TYPE "UDT_Motion_Point_IAI"
VERSION : 0.1
// =================================================================================
// UDT_Recipe_Final.scl
// Version: Final
//
// Description:
// Final, definitive recipe structure based on deep code analysis.
// - Axis names and mapping are CORRECT.
// - Position names are simple and numeric (Position_01, Position_02, ...)
//   to provide a safe, 1-to-1 mapping with the axis driver's position array.
//   This structure can be used to build a descriptive HMI.
// =================================================================================
// =================================================================================
// BASE TYPES for Motion Points
// =================================================================================
   STRUCT
      Pos : Real;   //  Target Position (um/pulse)
      Vel : Int;   //  Target Velocity (mm/s or %)
   END_STRUCT;

END_TYPE

TYPE "UDT_Motion_Point_V90"
VERSION : 0.1
   STRUCT
      Pos : DInt;   //  Target Position (mm/deg)
      Vel : Int;   //  Target Velocity (mm/s or rpm)
   END_STRUCT;

END_TYPE

TYPE "UDT_Recipe_PressCurve"
VERSION : 0.1
// NOTE: UDT_Recipe_PressCurve and UDT_Recipe_ATEQ are assumed to exist from original project files.
// =================================================================================
// MAIN RECIPE UDT - FINAL VERSION
// =================================================================================
   STRUCT
      StartPos_UL : Real;
      StartPos_LL : Real;
      StartForce_UL : Real;
      StartForce_LL : Real;
      MiddlePos_UL : Real;
      MiddlePos_LL : Real;
      MiddleForce_UL : Real;
      MiddleForce_LL : Real;
      FinalPos_UL : Real;
      FinalPos_LL : Real;
      FinalForce_UL : Real;
      FinalForce_LL : Real;
      ProgramNum : Int;
   END_STRUCT;

END_TYPE

TYPE "UDT_Gripper_Fixture_Codes"
VERSION : 0.1
// =================================================================================
// OTHER UDTs (Grippers, Process, etc. - Unchanged from previous correct versions)
// =================================================================================
   STRUCT
      "JAW TOOLING LEFT" : String[128];
      "JAW TOOLING RIGHT" : String[128];
      "SHAFT CLAMPING LEFT" : String[128];
      "SHAFT CLAMPING RIGHT" : String[128];
   END_STRUCT;

END_TYPE

TYPE "UDT_IAI_Axis_Positions"
VERSION : 0.1
// =================================================================================
// POSITION SETS - Mirroring the Axis Driver's Position Array
// =================================================================================
   STRUCT
      Position : Array[1..20] of "UDT_Motion_Point_IAI";
   END_STRUCT;

END_TYPE

TYPE "UDT_V90_Axis_Positions"
VERSION : 0.1
   STRUCT
      Position : Array[1..20] of "UDT_Motion_Point_V90";
   END_STRUCT;

END_TYPE

TYPE "UDT_OP10_Recipe_type"
VERSION : 0.1
   STRUCT
      Header : Struct   // Information about recipe
         RecipeName : String[50];   // name of product
         RecipeID : USInt;   // number of product for sig exch. and other processes
         "Version" : UInt;   // version of update that structure
         LastModified {InstructionName := 'DTL'; LibVersion := '1.0'} : DTL;   // time of last modifiacation
         PartType : String[28];   // second name for product - additional one
         PartTypeRecordNr : Int;   // PartType Record number same like recipi id for future sig exchanges etc
      END_STRUCT;
      Process : Struct   // Important process parameters how should machine act
         Timers : Struct   // Definition of times for processess
            Delay_glue_init_start : Time := t#2s;
            Delay_Medium : Time;
            Delay_Long : Time;
            Cylinder_ActTime : Time;
         END_STRUCT;
         Limits : Struct   // limitations of the values
            RetryLimit : Int;
         END_STRUCT;
         Press : Struct   // parameters for the kistler press devices
            B1_Program : Int;
            B2_Program : Int;
            Curve : "UDT_Recipe_PressCurve";
         END_STRUCT;
         Vision : Struct   // camera system programs numbers
            CGlueShaftIV3_Progs : Array[1..4] of Word;
            CGlueMagnetIV3_Prog : Word;
            CGlueProgram : Int;
         END_STRUCT;
      END_STRUCT;
      "Tooling Code" : Struct   // QR CODES OF THE TOOLING FOR THE RECIPE
         A1_Table : Array[1..8] of String[128];
         A2_Table : Array[1..8] of String[128];   //  ... other fixture codes Descriptive Gripper Fixture Codes
         ROB1_Shaft_Handling_Robot : Struct   //  R1
            Gripper : "UDT_Gripper_Fixture_Codes";
         END_STRUCT;
         ROB2_Main_Assembly_Robot : Struct   //  R2
            Gripper : "UDT_Gripper_Fixture_Codes";
         END_STRUCT;
         ROB3_Unloading_Robot : Struct   //  R3
            Gripper : "UDT_Gripper_Fixture_Codes";
         END_STRUCT;
         A1_Fixtures : Struct
            A1RingUnloadingFixtureCode : String[128];
            E1LoadingNGFixtureCode : String[128];
            ShaftScanFixtureCode : String[128];
            B1PressFixtureCode : String[128];
            CGlueFixtureCode : String[128];
            B1PressCylFixtureCode : String[128];
         END_STRUCT;
         A2_Fixtures : Struct
            A2RingUnloadingFixtureCode : String[128];
            E2UnloadingNGFixtureCode : String[128];
            B2PressFixtureCode : String[128];
            CGlueNGFixtureCode : String[128];
            B2PressCylFixtureCode : String[128];
         END_STRUCT;
      END_STRUCT;
      Motion : Struct   // ALL SERVO DRIVES PARAMETERS
         Gluing_Nozzle_Z : "UDT_IAI_Axis_Positions";   //  Physical Axis: IAI_A1
         Gluing_Nozzle_X : "UDT_IAI_Axis_Positions";   //  Physical Axis: IAI_A2
         Gluing_Nozzle_Y : "UDT_IAI_Axis_Positions";   //  Physical Axis: IAI_A3 CORRECTED V90 Axis Functions (from user)
         Ring_Turntable_Axis_1 : "UDT_V90_Axis_Positions";   //  Physical Axis: V90_A1
         Shaft_Scan_Turntable_Axis : "UDT_V90_Axis_Positions";   //  Physical Axis: V90_A2
         Gluing_Rotary_Jig_Axis : "UDT_V90_Axis_Positions";   //  Physical Axis: V90_A3
         Ring_Turntable_Axis_2 : "UDT_V90_Axis_Positions";   //  Physical Axis: V90_A4
      END_STRUCT;
   END_STRUCT;

END_TYPE

DATA_BLOCK "DB_ALL_PROCESS_PARAMETERS"
{ S7_Optimized_Access := 'TRUE' }
VERSION : 0.1
NON_RETAIN
   VAR RETAIN
      "Choosen Recipe Number" : Bool;
      ACTUAL_CHOOSEN_TYPE { S7_SetPoint := 'False'} : "UDT_OP10_Recipe_type";   // THERE IS ASCTUAL DATA READED OUT FROM LIBRARY OF 20 TYPES BELOW
      PRODUCT_TYPE { S7_SetPoint := 'False'} : Array[1..10] of "UDT_OP10_Recipe_type";   // PACK OF TWENTY DIFFERENT TYPES PRODUCT AND THEIR PARAMETERS FOR THE PROCESS
   END_VAR


BEGIN
   ACTUAL_CHOOSEN_TYPE.Header.RecipeName := 'produkt 1';
   ACTUAL_CHOOSEN_TYPE.Header.RecipeID := 2;
   ACTUAL_CHOOSEN_TYPE.Header."Version" := 19629;
   ACTUAL_CHOOSEN_TYPE.Header.LastModified.YEAR := 2026;
   ACTUAL_CHOOSEN_TYPE.Header.LastModified.MONTH := 1;
   ACTUAL_CHOOSEN_TYPE.Header.LastModified.DAY := 17;
   ACTUAL_CHOOSEN_TYPE.Header.LastModified.WEEKDAY := 7;
   ACTUAL_CHOOSEN_TYPE.Header.LastModified.HOUR := 4;
   ACTUAL_CHOOSEN_TYPE.Header.LastModified.MINUTE := 23;
   ACTUAL_CHOOSEN_TYPE.Header.LastModified.SECOND := 27;
   ACTUAL_CHOOSEN_TYPE.Header.LastModified.NANOSECOND := 501000000;
   ACTUAL_CHOOSEN_TYPE.Header.LastModified := DTL#2026-01-17-04:23:27.501;
   ACTUAL_CHOOSEN_TYPE.Header.PartType := 'additional  name';
   ACTUAL_CHOOSEN_TYPE.Header.PartTypeRecordNr := 0;
   ACTUAL_CHOOSEN_TYPE.Process.Timers.Delay_glue_init_start := T#2S;
   ACTUAL_CHOOSEN_TYPE.Process.Timers.Delay_Medium := T#600MS;
   ACTUAL_CHOOSEN_TYPE.Process.Timers.Delay_Long := T#2S;
   ACTUAL_CHOOSEN_TYPE.Process.Timers.Cylinder_ActTime := T#6S;
   ACTUAL_CHOOSEN_TYPE.Process.Limits.RetryLimit := 3;
   ACTUAL_CHOOSEN_TYPE.Process.Press.B1_Program := 1;
   ACTUAL_CHOOSEN_TYPE.Process.Press.B2_Program := 1;
   ACTUAL_CHOOSEN_TYPE.Process.Press.Curve.StartPos_UL := 0.0;
   ACTUAL_CHOOSEN_TYPE.Process.Press.Curve.StartPos_LL := 0.0;
   ACTUAL_CHOOSEN_TYPE.Process.Press.Curve.StartForce_UL := 0.0;
   ACTUAL_CHOOSEN_TYPE.Process.Press.Curve.StartForce_LL := 0.0;
   ACTUAL_CHOOSEN_TYPE.Process.Press.Curve.MiddlePos_UL := 0.0;
   ACTUAL_CHOOSEN_TYPE.Process.Press.Curve.MiddlePos_LL := 0.0;
   ACTUAL_CHOOSEN_TYPE.Process.Press.Curve.MiddleForce_UL := 0.0;
   ACTUAL_CHOOSEN_TYPE.Process.Press.Curve.MiddleForce_LL := 0.0;
   ACTUAL_CHOOSEN_TYPE.Process.Press.Curve.FinalPos_UL := 0.0;
   ACTUAL_CHOOSEN_TYPE.Process.Press.Curve.FinalPos_LL := 0.0;
   ACTUAL_CHOOSEN_TYPE.Process.Press.Curve.FinalForce_UL := 0.0;
   ACTUAL_CHOOSEN_TYPE.Process.Press.Curve.FinalForce_LL := 0.0;
   ACTUAL_CHOOSEN_TYPE.Process.Press.Curve.ProgramNum := 0;
   ACTUAL_CHOOSEN_TYPE.Process.Vision.CGlueShaftIV3_Progs[1] := 16#0001;
   ACTUAL_CHOOSEN_TYPE.Process.Vision.CGlueShaftIV3_Progs[2] := 16#0002;
   ACTUAL_CHOOSEN_TYPE.Process.Vision.CGlueShaftIV3_Progs[3] := 16#0003;
   ACTUAL_CHOOSEN_TYPE.Process.Vision.CGlueShaftIV3_Progs[4] := 16#0004;
   ACTUAL_CHOOSEN_TYPE.Process.Vision.CGlueMagnetIV3_Prog := 16#0001;
   ACTUAL_CHOOSEN_TYPE.Process.Vision.CGlueProgram := 1;
   ACTUAL_CHOOSEN_TYPE."Tooling Code".A1_Table[1] := 'SZ23055-OP010-E-Compressor-ring1 Loading tooling-1';
   ACTUAL_CHOOSEN_TYPE."Tooling Code".A1_Table[2] := 'SZ23055-OP010-E-Compressor-ring1 Loading tooling-2';
   ACTUAL_CHOOSEN_TYPE."Tooling Code".A1_Table[3] := 'SZ23055-OP010-E-Compressor-ring1 Loading tooling-3';
   ACTUAL_CHOOSEN_TYPE."Tooling Code".A1_Table[4] := 'SZ23055-OP010-E-Compressor-ring1 Loading tooling-4';
   ACTUAL_CHOOSEN_TYPE."Tooling Code".A1_Table[5] := 'SZ23055-OP010-E-Compressor-ring1 Loading tooling-5';
   ACTUAL_CHOOSEN_TYPE."Tooling Code".A1_Table[6] := 'SZ23055-OP010-E-Compressor-ring1 Loading tooling-6';
   ACTUAL_CHOOSEN_TYPE."Tooling Code".A1_Table[7] := 'SZ23055-OP010-E-Compressor-ring1 Loading tooling-7';
   ACTUAL_CHOOSEN_TYPE."Tooling Code".A1_Table[8] := 'SZ23055-OP010-E-Compressor-ring1 Loading tooling-8';
   ACTUAL_CHOOSEN_TYPE."Tooling Code".A2_Table[1] := 'SZ23055-OP010-E-Compresspr-ring1 cutting tool';
   ACTUAL_CHOOSEN_TYPE."Tooling Code".A2_Table[2] := 'SZ23055-OP010-E-Compressor-Left NG tooling-1';
   ACTUAL_CHOOSEN_TYPE."Tooling Code".A2_Table[3] := 'SZ23055-OP010-E-Compressor-shaft Rotating scanning tooling-1';
   ACTUAL_CHOOSEN_TYPE."Tooling Code".A2_Table[4] := 'SZ23055-OP010-E-Compressor-ring1 Below Positioning fixture -1';
   ACTUAL_CHOOSEN_TYPE."Tooling Code".A2_Table[5] := 'SZ23055-OP010-E-Compressor-Point adhesive tooling-1';
   ACTUAL_CHOOSEN_TYPE."Tooling Code".A2_Table[6] := 'SZ23055-OP010-E-Compressor-ring1 Upper pressing fixture-1';
   ACTUAL_CHOOSEN_TYPE."Tooling Code".A2_Table[7] := 'SZ23055-OP010-E-Compresspr-ring2 cutting tool';
   ACTUAL_CHOOSEN_TYPE."Tooling Code".A2_Table[8] := 'SZ23055-OP010-E-Compressor-Right NG tooling-1';
   ACTUAL_CHOOSEN_TYPE."Tooling Code".ROB1_Shaft_Handling_Robot.Gripper."JAW TOOLING LEFT" := 'SZ23055-OP010-E-Compressor-robot1 ring1 Left clamping jaw tooling-1';
   ACTUAL_CHOOSEN_TYPE."Tooling Code".ROB1_Shaft_Handling_Robot.Gripper."JAW TOOLING RIGHT" := 'SZ23055-OP010-E-Compressor-robot1 ring1 Right clamping jaw tooling-2';
   ACTUAL_CHOOSEN_TYPE."Tooling Code".ROB1_Shaft_Handling_Robot.Gripper."SHAFT CLAMPING LEFT" := 'SZ23055-OP010-E-Compressor-robot1 shaft Left clamping jaw tooling-1';
   ACTUAL_CHOOSEN_TYPE."Tooling Code".ROB1_Shaft_Handling_Robot.Gripper."SHAFT CLAMPING RIGHT" := 'SZ23055-OP010-E-Compressor-robot1 shaft Right clamping jaw tooling-2';
   ACTUAL_CHOOSEN_TYPE."Tooling Code".ROB2_Main_Assembly_Robot.Gripper."JAW TOOLING LEFT" := 'SZ23055-OP010-E-Compressor-robot2 shaft Right clamping jaw tooling-2';
   ACTUAL_CHOOSEN_TYPE."Tooling Code".ROB2_Main_Assembly_Robot.Gripper."JAW TOOLING RIGHT" := 'SZ23055-OP010-E-Compressor-robot2 shaft Left clamping jaw tooling-1';
   ACTUAL_CHOOSEN_TYPE."Tooling Code".ROB2_Main_Assembly_Robot.Gripper."SHAFT CLAMPING LEFT" := 'SZ23055-OP010-E-Compressor-robot2 magnet Right clamping jaw tooling-2';
   ACTUAL_CHOOSEN_TYPE."Tooling Code".ROB2_Main_Assembly_Robot.Gripper."SHAFT CLAMPING RIGHT" := 'SZ23055-OP010-E-Compressor-robot2 magnet Right clamping jaw tooling-2';
   ACTUAL_CHOOSEN_TYPE."Tooling Code".ROB3_Unloading_Robot.Gripper."JAW TOOLING LEFT" := 'SZ23055-OP010-E-Compressor-robot3 ring2 Right clamping jaw tooling-2';
   ACTUAL_CHOOSEN_TYPE."Tooling Code".ROB3_Unloading_Robot.Gripper."JAW TOOLING RIGHT" := 'SZ23055-OP010-E-Compressor-robot3 ring2 Left clamping jaw tooling-1';
   ACTUAL_CHOOSEN_TYPE."Tooling Code".ROB3_Unloading_Robot.Gripper."SHAFT CLAMPING LEFT" := 'SZ23055-OP010-E-Compressor-robot3 shaft Left clamping jaw tooling-1';
   ACTUAL_CHOOSEN_TYPE."Tooling Code".ROB3_Unloading_Robot.Gripper."SHAFT CLAMPING RIGHT" := 'SZ23055-OP010-E-Compressor-robot3 shaft Right clamping jaw tooling-2';
   ACTUAL_CHOOSEN_TYPE."Tooling Code".A1_Fixtures.A1RingUnloadingFixtureCode := 'SZ23055-OP010-E-Compresspr-ring1 cutting tool';
   ACTUAL_CHOOSEN_TYPE."Tooling Code".A1_Fixtures.E1LoadingNGFixtureCode := 'SZ23055-OP010-E-Compressor-Left NG tooling-1';
   ACTUAL_CHOOSEN_TYPE."Tooling Code".A1_Fixtures.ShaftScanFixtureCode := 'SZ23055-OP010-E-Compressor-shaft Rotating scanning tooling-1';
   ACTUAL_CHOOSEN_TYPE."Tooling Code".A1_Fixtures.B1PressFixtureCode := 'SZ23055-OP010-E-Compressor-ring1 Below Positioning fixture -1';
   ACTUAL_CHOOSEN_TYPE."Tooling Code".A1_Fixtures.CGlueFixtureCode := 'SZ23055-OP010-E-Compressor-Point adhesive tooling-1';
   ACTUAL_CHOOSEN_TYPE."Tooling Code".A1_Fixtures.B1PressCylFixtureCode := 'SZ23055-OP010-E-Compressor-ring1 Upper pressing fixture-1';
   ACTUAL_CHOOSEN_TYPE."Tooling Code".A2_Fixtures.A2RingUnloadingFixtureCode := 'SZ23055-OP010-E-Compresspr-ring2 cutting tool';
   ACTUAL_CHOOSEN_TYPE."Tooling Code".A2_Fixtures.E2UnloadingNGFixtureCode := 'SZ23055-OP010-E-Compressor-Right NG tooling-1';
   ACTUAL_CHOOSEN_TYPE."Tooling Code".A2_Fixtures.B2PressFixtureCode := 'SZ23055-OP010-E-Compressor-ring2 Below Positioning fixture -1';
   ACTUAL_CHOOSEN_TYPE."Tooling Code".A2_Fixtures.CGlueNGFixtureCode := 'SZ23055-OP010-E-Compressor-NG middle shift tooling-1';
   ACTUAL_CHOOSEN_TYPE."Tooling Code".A2_Fixtures.B2PressCylFixtureCode := 'SZ23055-OP010-E-Compressor-ring2 Upper pressing fixture-1';
   PRODUCT_TYPE[1].Header.RecipeName := 'produkt 1';
   PRODUCT_TYPE[1].Header.RecipeID := 1;
   PRODUCT_TYPE[1].Header."Version" := 1;
   PRODUCT_TYPE[1].Header.LastModified.YEAR := 2026;
   PRODUCT_TYPE[1].Header.LastModified.MONTH := 1;
   PRODUCT_TYPE[1].Header.LastModified.DAY := 17;
   PRODUCT_TYPE[1].Header.LastModified.WEEKDAY := 7;
   PRODUCT_TYPE[1].Header.LastModified.HOUR := 4;
   PRODUCT_TYPE[1].Header.LastModified.MINUTE := 23;
   PRODUCT_TYPE[1].Header.LastModified.SECOND := 27;
   PRODUCT_TYPE[1].Header.LastModified.NANOSECOND := 501000000;
   PRODUCT_TYPE[1].Header.LastModified := DTL#2026-01-17-04:23:27.501;
   PRODUCT_TYPE[1].Header.PartType := 'additional  name';
   PRODUCT_TYPE[1].Header.PartTypeRecordNr := 0;
   PRODUCT_TYPE[1].Process.Timers.Delay_glue_init_start := T#2S;
   PRODUCT_TYPE[1].Process.Timers.Delay_Medium := T#600MS;
   PRODUCT_TYPE[1].Process.Timers.Delay_Long := T#2S;
   PRODUCT_TYPE[1].Process.Timers.Cylinder_ActTime := T#6S;
   PRODUCT_TYPE[1].Process.Limits.RetryLimit := 3;
   PRODUCT_TYPE[1].Process.Press.B1_Program := 1;
   PRODUCT_TYPE[1].Process.Press.B2_Program := 1;
   PRODUCT_TYPE[1].Process.Press.Curve.StartPos_UL := 0.0;
   PRODUCT_TYPE[1].Process.Press.Curve.StartPos_LL := 0.0;
   PRODUCT_TYPE[1].Process.Press.Curve.StartForce_UL := 0.0;
   PRODUCT_TYPE[1].Process.Press.Curve.StartForce_LL := 0.0;
   PRODUCT_TYPE[1].Process.Press.Curve.MiddlePos_UL := 0.0;
   PRODUCT_TYPE[1].Process.Press.Curve.MiddlePos_LL := 0.0;
   PRODUCT_TYPE[1].Process.Press.Curve.MiddleForce_UL := 0.0;
   PRODUCT_TYPE[1].Process.Press.Curve.MiddleForce_LL := 0.0;
   PRODUCT_TYPE[1].Process.Press.Curve.FinalPos_UL := 0.0;
   PRODUCT_TYPE[1].Process.Press.Curve.FinalPos_LL := 0.0;
   PRODUCT_TYPE[1].Process.Press.Curve.FinalForce_UL := 0.0;
   PRODUCT_TYPE[1].Process.Press.Curve.FinalForce_LL := 0.0;
   PRODUCT_TYPE[1].Process.Press.Curve.ProgramNum := 0;
   PRODUCT_TYPE[1].Process.Vision.CGlueShaftIV3_Progs[1] := 16#0001;
   PRODUCT_TYPE[1].Process.Vision.CGlueShaftIV3_Progs[2] := 16#0002;
   PRODUCT_TYPE[1].Process.Vision.CGlueShaftIV3_Progs[3] := 16#0003;
   PRODUCT_TYPE[1].Process.Vision.CGlueShaftIV3_Progs[4] := 16#0004;
   PRODUCT_TYPE[1].Process.Vision.CGlueMagnetIV3_Prog := 16#0001;
   PRODUCT_TYPE[1].Process.Vision.CGlueProgram := 1;
   PRODUCT_TYPE[1]."Tooling Code".A1_Table[1] := 'SZ23055-OP010-E-Compressor-ring1 Loading tooling-1';
   PRODUCT_TYPE[1]."Tooling Code".A1_Table[2] := 'SZ23055-OP010-E-Compressor-ring1 Loading tooling-2';
   PRODUCT_TYPE[1]."Tooling Code".A1_Table[3] := 'SZ23055-OP010-E-Compressor-ring1 Loading tooling-3';
   PRODUCT_TYPE[1]."Tooling Code".A1_Table[4] := 'SZ23055-OP010-E-Compressor-ring1 Loading tooling-4';
   PRODUCT_TYPE[1]."Tooling Code".A1_Table[5] := 'SZ23055-OP010-E-Compressor-ring1 Loading tooling-5';
   PRODUCT_TYPE[1]."Tooling Code".A1_Table[6] := 'SZ23055-OP010-E-Compressor-ring1 Loading tooling-6';
   PRODUCT_TYPE[1]."Tooling Code".A1_Table[7] := 'SZ23055-OP010-E-Compressor-ring1 Loading tooling-7';
   PRODUCT_TYPE[1]."Tooling Code".A1_Table[8] := 'SZ23055-OP010-E-Compressor-ring1 Loading tooling-8';
   PRODUCT_TYPE[1]."Tooling Code".A2_Table[1] := 'SZ23055-OP010-E-Compresspr-ring1 cutting tool';
   PRODUCT_TYPE[1]."Tooling Code".A2_Table[2] := 'SZ23055-OP010-E-Compressor-Left NG tooling-1';
   PRODUCT_TYPE[1]."Tooling Code".A2_Table[3] := 'SZ23055-OP010-E-Compressor-shaft Rotating scanning tooling-1';
   PRODUCT_TYPE[1]."Tooling Code".A2_Table[4] := 'SZ23055-OP010-E-Compressor-ring1 Below Positioning fixture -1';
   PRODUCT_TYPE[1]."Tooling Code".A2_Table[5] := 'SZ23055-OP010-E-Compressor-Point adhesive tooling-1';
   PRODUCT_TYPE[1]."Tooling Code".A2_Table[6] := 'SZ23055-OP010-E-Compressor-ring1 Upper pressing fixture-1';
   PRODUCT_TYPE[1]."Tooling Code".A2_Table[7] := 'SZ23055-OP010-E-Compresspr-ring2 cutting tool';
   PRODUCT_TYPE[1]."Tooling Code".A2_Table[8] := 'SZ23055-OP010-E-Compressor-Right NG tooling-1';
   PRODUCT_TYPE[1]."Tooling Code".ROB1_Shaft_Handling_Robot.Gripper."JAW TOOLING LEFT" := 'SZ23055-OP010-E-Compressor-robot1 ring1 Left clamping jaw tooling-1';
   PRODUCT_TYPE[1]."Tooling Code".ROB1_Shaft_Handling_Robot.Gripper."JAW TOOLING RIGHT" := 'SZ23055-OP010-E-Compressor-robot1 ring1 Right clamping jaw tooling-2';
   PRODUCT_TYPE[1]."Tooling Code".ROB1_Shaft_Handling_Robot.Gripper."SHAFT CLAMPING LEFT" := 'SZ23055-OP010-E-Compressor-robot1 shaft Left clamping jaw tooling-1';
   PRODUCT_TYPE[1]."Tooling Code".ROB1_Shaft_Handling_Robot.Gripper."SHAFT CLAMPING RIGHT" := 'SZ23055-OP010-E-Compressor-robot1 shaft Right clamping jaw tooling-2';
   PRODUCT_TYPE[1]."Tooling Code".ROB2_Main_Assembly_Robot.Gripper."JAW TOOLING LEFT" := 'SZ23055-OP010-E-Compressor-robot2 shaft Right clamping jaw tooling-2';
   PRODUCT_TYPE[1]."Tooling Code".ROB2_Main_Assembly_Robot.Gripper."JAW TOOLING RIGHT" := 'SZ23055-OP010-E-Compressor-robot2 shaft Left clamping jaw tooling-1';
   PRODUCT_TYPE[1]."Tooling Code".ROB2_Main_Assembly_Robot.Gripper."SHAFT CLAMPING LEFT" := 'SZ23055-OP010-E-Compressor-robot2 magnet Right clamping jaw tooling-2';
   PRODUCT_TYPE[1]."Tooling Code".ROB2_Main_Assembly_Robot.Gripper."SHAFT CLAMPING RIGHT" := 'SZ23055-OP010-E-Compressor-robot2 magnet Right clamping jaw tooling-2';
   PRODUCT_TYPE[1]."Tooling Code".ROB3_Unloading_Robot.Gripper."JAW TOOLING LEFT" := 'SZ23055-OP010-E-Compressor-robot3 ring2 Right clamping jaw tooling-2';
   PRODUCT_TYPE[1]."Tooling Code".ROB3_Unloading_Robot.Gripper."JAW TOOLING RIGHT" := 'SZ23055-OP010-E-Compressor-robot3 ring2 Left clamping jaw tooling-1';
   PRODUCT_TYPE[1]."Tooling Code".ROB3_Unloading_Robot.Gripper."SHAFT CLAMPING LEFT" := 'SZ23055-OP010-E-Compressor-robot3 shaft Left clamping jaw tooling-1';
   PRODUCT_TYPE[1]."Tooling Code".ROB3_Unloading_Robot.Gripper."SHAFT CLAMPING RIGHT" := 'SZ23055-OP010-E-Compressor-robot3 shaft Right clamping jaw tooling-2';
   PRODUCT_TYPE[1]."Tooling Code".A1_Fixtures.A1RingUnloadingFixtureCode := 'SZ23055-OP010-E-Compresspr-ring1 cutting tool';
   PRODUCT_TYPE[1]."Tooling Code".A1_Fixtures.E1LoadingNGFixtureCode := 'SZ23055-OP010-E-Compressor-Left NG tooling-1';
   PRODUCT_TYPE[1]."Tooling Code".A1_Fixtures.ShaftScanFixtureCode := 'SZ23055-OP010-E-Compressor-shaft Rotating scanning tooling-1';
   PRODUCT_TYPE[1]."Tooling Code".A1_Fixtures.B1PressFixtureCode := 'SZ23055-OP010-E-Compressor-ring1 Below Positioning fixture -1';
   PRODUCT_TYPE[1]."Tooling Code".A1_Fixtures.CGlueFixtureCode := 'SZ23055-OP010-E-Compressor-Point adhesive tooling-1';
   PRODUCT_TYPE[1]."Tooling Code".A1_Fixtures.B1PressCylFixtureCode := 'SZ23055-OP010-E-Compressor-ring1 Upper pressing fixture-1';
   PRODUCT_TYPE[1]."Tooling Code".A2_Fixtures.A2RingUnloadingFixtureCode := 'SZ23055-OP010-E-Compresspr-ring2 cutting tool';
   PRODUCT_TYPE[1]."Tooling Code".A2_Fixtures.E2UnloadingNGFixtureCode := 'SZ23055-OP010-E-Compressor-Right NG tooling-1';
   PRODUCT_TYPE[1]."Tooling Code".A2_Fixtures.B2PressFixtureCode := 'SZ23055-OP010-E-Compressor-ring2 Below Positioning fixture -1';
   PRODUCT_TYPE[1]."Tooling Code".A2_Fixtures.CGlueNGFixtureCode := 'SZ23055-OP010-E-Compressor-NG middle shift tooling-1';
   PRODUCT_TYPE[1]."Tooling Code".A2_Fixtures.B2PressCylFixtureCode := 'SZ23055-OP010-E-Compressor-ring2 Upper pressing fixture-1';
   PRODUCT_TYPE[2].Header.RecipeName := '';
   PRODUCT_TYPE[2].Header.RecipeID := 0;
   PRODUCT_TYPE[2].Header."Version" := 0;
   PRODUCT_TYPE[2].Header.LastModified.YEAR := 1970;
   PRODUCT_TYPE[2].Header.LastModified.MONTH := 1;
   PRODUCT_TYPE[2].Header.LastModified.DAY := 1;
   PRODUCT_TYPE[2].Header.LastModified.WEEKDAY := 5;
   PRODUCT_TYPE[2].Header.LastModified.HOUR := 0;
   PRODUCT_TYPE[2].Header.LastModified.MINUTE := 0;
   PRODUCT_TYPE[2].Header.LastModified.SECOND := 0;
   PRODUCT_TYPE[2].Header.LastModified.NANOSECOND := 0;
   PRODUCT_TYPE[2].Header.LastModified := DTL#1970-01-01-00:00:00;
   PRODUCT_TYPE[2].Header.PartType := '';
   PRODUCT_TYPE[2].Header.PartTypeRecordNr := 0;
   PRODUCT_TYPE[2].Process.Timers.Delay_glue_init_start := T#0MS;
   PRODUCT_TYPE[2].Process.Timers.Delay_Medium := T#0MS;
   PRODUCT_TYPE[2].Process.Timers.Delay_Long := T#0MS;
   PRODUCT_TYPE[2].Process.Timers.Cylinder_ActTime := T#0MS;
   PRODUCT_TYPE[2].Process.Limits.RetryLimit := 0;
   PRODUCT_TYPE[2].Process.Press.B1_Program := 0;
   PRODUCT_TYPE[2].Process.Press.B2_Program := 0;
   PRODUCT_TYPE[2].Process.Press.Curve.StartPos_UL := 0.0;
   PRODUCT_TYPE[2].Process.Press.Curve.StartPos_LL := 0.0;
   PRODUCT_TYPE[2].Process.Press.Curve.StartForce_UL := 0.0;
   PRODUCT_TYPE[2].Process.Press.Curve.StartForce_LL := 0.0;
   PRODUCT_TYPE[2].Process.Press.Curve.MiddlePos_UL := 0.0;
   PRODUCT_TYPE[2].Process.Press.Curve.MiddlePos_LL := 0.0;
   PRODUCT_TYPE[2].Process.Press.Curve.MiddleForce_UL := 0.0;
   PRODUCT_TYPE[2].Process.Press.Curve.MiddleForce_LL := 0.0;
   PRODUCT_TYPE[2].Process.Press.Curve.FinalPos_UL := 0.0;
   PRODUCT_TYPE[2].Process.Press.Curve.FinalPos_LL := 0.0;
   PRODUCT_TYPE[2].Process.Press.Curve.FinalForce_UL := 0.0;
   PRODUCT_TYPE[2].Process.Press.Curve.FinalForce_LL := 0.0;
   PRODUCT_TYPE[2].Process.Press.Curve.ProgramNum := 0;
   PRODUCT_TYPE[2].Process.Vision.CGlueShaftIV3_Progs[1] := 16#0000;
   PRODUCT_TYPE[2].Process.Vision.CGlueShaftIV3_Progs[2] := 16#0000;
   PRODUCT_TYPE[2].Process.Vision.CGlueShaftIV3_Progs[3] := 16#0000;
   PRODUCT_TYPE[2].Process.Vision.CGlueShaftIV3_Progs[4] := 16#0000;
   PRODUCT_TYPE[2].Process.Vision.CGlueMagnetIV3_Prog := 16#0000;
   PRODUCT_TYPE[2].Process.Vision.CGlueProgram := 0;
   PRODUCT_TYPE[2]."Tooling Code".A1_Table[1] := '';
   PRODUCT_TYPE[2]."Tooling Code".A1_Table[2] := '';
   PRODUCT_TYPE[2]."Tooling Code".A1_Table[3] := '';
   PRODUCT_TYPE[2]."Tooling Code".A1_Table[4] := '';
   PRODUCT_TYPE[2]."Tooling Code".A1_Table[5] := '';
   PRODUCT_TYPE[2]."Tooling Code".A1_Table[6] := '';
   PRODUCT_TYPE[2]."Tooling Code".A1_Table[7] := '';
   PRODUCT_TYPE[2]."Tooling Code".A1_Table[8] := '';
   PRODUCT_TYPE[2]."Tooling Code".A2_Table[1] := '';
   PRODUCT_TYPE[2]."Tooling Code".A2_Table[2] := '';
   PRODUCT_TYPE[2]."Tooling Code".A2_Table[3] := '';
   PRODUCT_TYPE[2]."Tooling Code".A2_Table[4] := '';
   PRODUCT_TYPE[2]."Tooling Code".A2_Table[5] := '';
   PRODUCT_TYPE[2]."Tooling Code".A2_Table[6] := '';
   PRODUCT_TYPE[2]."Tooling Code".A2_Table[7] := '';
   PRODUCT_TYPE[2]."Tooling Code".A2_Table[8] := '';
   PRODUCT_TYPE[2]."Tooling Code".ROB1_Shaft_Handling_Robot.Gripper."JAW TOOLING LEFT" := '';
   PRODUCT_TYPE[2]."Tooling Code".ROB1_Shaft_Handling_Robot.Gripper."JAW TOOLING RIGHT" := '';
   PRODUCT_TYPE[2]."Tooling Code".ROB1_Shaft_Handling_Robot.Gripper."SHAFT CLAMPING LEFT" := '';
   PRODUCT_TYPE[2]."Tooling Code".ROB1_Shaft_Handling_Robot.Gripper."SHAFT CLAMPING RIGHT" := '';
   PRODUCT_TYPE[2]."Tooling Code".ROB2_Main_Assembly_Robot.Gripper."JAW TOOLING LEFT" := '';
   PRODUCT_TYPE[2]."Tooling Code".ROB2_Main_Assembly_Robot.Gripper."JAW TOOLING RIGHT" := '';
   PRODUCT_TYPE[2]."Tooling Code".ROB2_Main_Assembly_Robot.Gripper."SHAFT CLAMPING LEFT" := '';
   PRODUCT_TYPE[2]."Tooling Code".ROB2_Main_Assembly_Robot.Gripper."SHAFT CLAMPING RIGHT" := '';
   PRODUCT_TYPE[2]."Tooling Code".ROB3_Unloading_Robot.Gripper."JAW TOOLING LEFT" := '';
   PRODUCT_TYPE[2]."Tooling Code".ROB3_Unloading_Robot.Gripper."JAW TOOLING RIGHT" := '';
   PRODUCT_TYPE[2]."Tooling Code".ROB3_Unloading_Robot.Gripper."SHAFT CLAMPING LEFT" := '';
   PRODUCT_TYPE[2]."Tooling Code".ROB3_Unloading_Robot.Gripper."SHAFT CLAMPING RIGHT" := '';
   PRODUCT_TYPE[2]."Tooling Code".A1_Fixtures.A1RingUnloadingFixtureCode := '';
   PRODUCT_TYPE[2]."Tooling Code".A1_Fixtures.E1LoadingNGFixtureCode := '';
   PRODUCT_TYPE[2]."Tooling Code".A1_Fixtures.ShaftScanFixtureCode := '';
   PRODUCT_TYPE[2]."Tooling Code".A1_Fixtures.B1PressFixtureCode := '';
   PRODUCT_TYPE[2]."Tooling Code".A1_Fixtures.CGlueFixtureCode := '';
   PRODUCT_TYPE[2]."Tooling Code".A1_Fixtures.B1PressCylFixtureCode := '';
   PRODUCT_TYPE[2]."Tooling Code".A2_Fixtures.A2RingUnloadingFixtureCode := '';
   PRODUCT_TYPE[2]."Tooling Code".A2_Fixtures.E2UnloadingNGFixtureCode := '';
   PRODUCT_TYPE[2]."Tooling Code".A2_Fixtures.B2PressFixtureCode := '';
   PRODUCT_TYPE[2]."Tooling Code".A2_Fixtures.CGlueNGFixtureCode := '';
   PRODUCT_TYPE[2]."Tooling Code".A2_Fixtures.B2PressCylFixtureCode := '';
   PRODUCT_TYPE[3].Header.RecipeName := 'produkt 1';
   PRODUCT_TYPE[3].Header.RecipeID := 1;
   PRODUCT_TYPE[3].Header."Version" := 1;
   PRODUCT_TYPE[3].Header.LastModified.YEAR := 2026;
   PRODUCT_TYPE[3].Header.LastModified.MONTH := 1;
   PRODUCT_TYPE[3].Header.LastModified.DAY := 17;
   PRODUCT_TYPE[3].Header.LastModified.WEEKDAY := 7;
   PRODUCT_TYPE[3].Header.LastModified.HOUR := 4;
   PRODUCT_TYPE[3].Header.LastModified.MINUTE := 23;
   PRODUCT_TYPE[3].Header.LastModified.SECOND := 27;
   PRODUCT_TYPE[3].Header.LastModified.NANOSECOND := 501000000;
   PRODUCT_TYPE[3].Header.LastModified := DTL#2026-01-17-04:23:27.501;
   PRODUCT_TYPE[3].Header.PartType := 'additional  name';
   PRODUCT_TYPE[3].Header.PartTypeRecordNr := 0;
   PRODUCT_TYPE[3].Process.Timers.Delay_glue_init_start := T#300MS;
   PRODUCT_TYPE[3].Process.Timers.Delay_Medium := T#600MS;
   PRODUCT_TYPE[3].Process.Timers.Delay_Long := T#2S;
   PRODUCT_TYPE[3].Process.Timers.Cylinder_ActTime := T#6S;
   PRODUCT_TYPE[3].Process.Limits.RetryLimit := 3;
   PRODUCT_TYPE[3].Process.Press.B1_Program := 1;
   PRODUCT_TYPE[3].Process.Press.B2_Program := 1;
   PRODUCT_TYPE[3].Process.Press.Curve.StartPos_UL := 0.0;
   PRODUCT_TYPE[3].Process.Press.Curve.StartPos_LL := 0.0;
   PRODUCT_TYPE[3].Process.Press.Curve.StartForce_UL := 0.0;
   PRODUCT_TYPE[3].Process.Press.Curve.StartForce_LL := 0.0;
   PRODUCT_TYPE[3].Process.Press.Curve.MiddlePos_UL := 0.0;
   PRODUCT_TYPE[3].Process.Press.Curve.MiddlePos_LL := 0.0;
   PRODUCT_TYPE[3].Process.Press.Curve.MiddleForce_UL := 0.0;
   PRODUCT_TYPE[3].Process.Press.Curve.MiddleForce_LL := 0.0;
   PRODUCT_TYPE[3].Process.Press.Curve.FinalPos_UL := 0.0;
   PRODUCT_TYPE[3].Process.Press.Curve.FinalPos_LL := 0.0;
   PRODUCT_TYPE[3].Process.Press.Curve.FinalForce_UL := 0.0;
   PRODUCT_TYPE[3].Process.Press.Curve.FinalForce_LL := 0.0;
   PRODUCT_TYPE[3].Process.Press.Curve.ProgramNum := 0;
   PRODUCT_TYPE[3].Process.Vision.CGlueShaftIV3_Progs[1] := 16#0001;
   PRODUCT_TYPE[3].Process.Vision.CGlueShaftIV3_Progs[2] := 16#0002;
   PRODUCT_TYPE[3].Process.Vision.CGlueShaftIV3_Progs[3] := 16#0003;
   PRODUCT_TYPE[3].Process.Vision.CGlueShaftIV3_Progs[4] := 16#0004;
   PRODUCT_TYPE[3].Process.Vision.CGlueMagnetIV3_Prog := 16#0001;
   PRODUCT_TYPE[3].Process.Vision.CGlueProgram := 1;
   PRODUCT_TYPE[3]."Tooling Code".A1_Table[1] := 'SZ23055-OP010-E-Compressor-ring1 Loading tooling-1';
   PRODUCT_TYPE[3]."Tooling Code".A1_Table[2] := 'SZ23055-OP010-E-Compressor-ring1 Loading tooling-2';
   PRODUCT_TYPE[3]."Tooling Code".A1_Table[3] := 'SZ23055-OP010-E-Compressor-ring1 Loading tooling-3';
   PRODUCT_TYPE[3]."Tooling Code".A1_Table[4] := 'SZ23055-OP010-E-Compressor-ring1 Loading tooling-4';
   PRODUCT_TYPE[3]."Tooling Code".A1_Table[5] := 'SZ23055-OP010-E-Compressor-ring1 Loading tooling-5';
   PRODUCT_TYPE[3]."Tooling Code".A1_Table[6] := 'SZ23055-OP010-E-Compressor-ring1 Loading tooling-6';
   PRODUCT_TYPE[3]."Tooling Code".A1_Table[7] := 'SZ23055-OP010-E-Compressor-ring1 Loading tooling-7';
   PRODUCT_TYPE[3]."Tooling Code".A1_Table[8] := 'SZ23055-OP010-E-Compressor-ring1 Loading tooling-8';
   PRODUCT_TYPE[3]."Tooling Code".A2_Table[1] := 'SZ23055-OP010-E-Compresspr-ring1 cutting tool';
   PRODUCT_TYPE[3]."Tooling Code".A2_Table[2] := 'SZ23055-OP010-E-Compressor-Left NG tooling-1';
   PRODUCT_TYPE[3]."Tooling Code".A2_Table[3] := 'SZ23055-OP010-E-Compressor-shaft Rotating scanning tooling-1';
   PRODUCT_TYPE[3]."Tooling Code".A2_Table[4] := 'SZ23055-OP010-E-Compressor-ring1 Below Positioning fixture -1';
   PRODUCT_TYPE[3]."Tooling Code".A2_Table[5] := 'SZ23055-OP010-E-Compressor-Point adhesive tooling-1';
   PRODUCT_TYPE[3]."Tooling Code".A2_Table[6] := 'SZ23055-OP010-E-Compressor-ring1 Upper pressing fixture-1';
   PRODUCT_TYPE[3]."Tooling Code".A2_Table[7] := 'SZ23055-OP010-E-Compresspr-ring2 cutting tool';
   PRODUCT_TYPE[3]."Tooling Code".A2_Table[8] := 'SZ23055-OP010-E-Compressor-Right NG tooling-1';
   PRODUCT_TYPE[3]."Tooling Code".ROB1_Shaft_Handling_Robot.Gripper."JAW TOOLING LEFT" := 'SZ23055-OP010-E-Compressor-robot1 ring1 Left clamping jaw tooling-1';
   PRODUCT_TYPE[3]."Tooling Code".ROB1_Shaft_Handling_Robot.Gripper."JAW TOOLING RIGHT" := 'SZ23055-OP010-E-Compressor-robot1 ring1 Right clamping jaw tooling-2';
   PRODUCT_TYPE[3]."Tooling Code".ROB1_Shaft_Handling_Robot.Gripper."SHAFT CLAMPING LEFT" := 'SZ23055-OP010-E-Compressor-robot1 shaft Left clamping jaw tooling-1';
   PRODUCT_TYPE[3]."Tooling Code".ROB1_Shaft_Handling_Robot.Gripper."SHAFT CLAMPING RIGHT" := 'SZ23055-OP010-E-Compressor-robot1 shaft Right clamping jaw tooling-2';
   PRODUCT_TYPE[3]."Tooling Code".ROB2_Main_Assembly_Robot.Gripper."JAW TOOLING LEFT" := 'SZ23055-OP010-E-Compressor-robot2 shaft Right clamping jaw tooling-2';
   PRODUCT_TYPE[3]."Tooling Code".ROB2_Main_Assembly_Robot.Gripper."JAW TOOLING RIGHT" := 'SZ23055-OP010-E-Compressor-robot2 shaft Left clamping jaw tooling-1';
   PRODUCT_TYPE[3]."Tooling Code".ROB2_Main_Assembly_Robot.Gripper."SHAFT CLAMPING LEFT" := 'SZ23055-OP010-E-Compressor-robot2 magnet Right clamping jaw tooling-2';
   PRODUCT_TYPE[3]."Tooling Code".ROB2_Main_Assembly_Robot.Gripper."SHAFT CLAMPING RIGHT" := 'SZ23055-OP010-E-Compressor-robot2 magnet Right clamping jaw tooling-2';
   PRODUCT_TYPE[3]."Tooling Code".ROB3_Unloading_Robot.Gripper."JAW TOOLING LEFT" := 'SZ23055-OP010-E-Compressor-robot3 ring2 Right clamping jaw tooling-2';
   PRODUCT_TYPE[3]."Tooling Code".ROB3_Unloading_Robot.Gripper."JAW TOOLING RIGHT" := 'SZ23055-OP010-E-Compressor-robot3 ring2 Left clamping jaw tooling-1';
   PRODUCT_TYPE[3]."Tooling Code".ROB3_Unloading_Robot.Gripper."SHAFT CLAMPING LEFT" := 'SZ23055-OP010-E-Compressor-robot3 shaft Left clamping jaw tooling-1';
   PRODUCT_TYPE[3]."Tooling Code".ROB3_Unloading_Robot.Gripper."SHAFT CLAMPING RIGHT" := 'SZ23055-OP010-E-Compressor-robot3 shaft Right clamping jaw tooling-2';
   PRODUCT_TYPE[3]."Tooling Code".A1_Fixtures.A1RingUnloadingFixtureCode := 'SZ23055-OP010-E-Compresspr-ring1 cutting tool';
   PRODUCT_TYPE[3]."Tooling Code".A1_Fixtures.E1LoadingNGFixtureCode := 'SZ23055-OP010-E-Compressor-Left NG tooling-1';
   PRODUCT_TYPE[3]."Tooling Code".A1_Fixtures.ShaftScanFixtureCode := 'SZ23055-OP010-E-Compressor-shaft Rotating scanning tooling-1';
   PRODUCT_TYPE[3]."Tooling Code".A1_Fixtures.B1PressFixtureCode := 'SZ23055-OP010-E-Compressor-ring1 Below Positioning fixture -1';
   PRODUCT_TYPE[3]."Tooling Code".A1_Fixtures.CGlueFixtureCode := 'SZ23055-OP010-E-Compressor-Point adhesive tooling-1';
   PRODUCT_TYPE[3]."Tooling Code".A1_Fixtures.B1PressCylFixtureCode := 'SZ23055-OP010-E-Compressor-ring1 Upper pressing fixture-1';
   PRODUCT_TYPE[3]."Tooling Code".A2_Fixtures.A2RingUnloadingFixtureCode := 'SZ23055-OP010-E-Compresspr-ring2 cutting tool';
   PRODUCT_TYPE[3]."Tooling Code".A2_Fixtures.E2UnloadingNGFixtureCode := 'SZ23055-OP010-E-Compressor-Right NG tooling-1';
   PRODUCT_TYPE[3]."Tooling Code".A2_Fixtures.B2PressFixtureCode := 'SZ23055-OP010-E-Compressor-ring2 Below Positioning fixture -1';
   PRODUCT_TYPE[3]."Tooling Code".A2_Fixtures.CGlueNGFixtureCode := 'SZ23055-OP010-E-Compressor-NG middle shift tooling-1';
   PRODUCT_TYPE[3]."Tooling Code".A2_Fixtures.B2PressCylFixtureCode := 'SZ23055-OP010-E-Compressor-ring2 Upper pressing fixture-1';
   PRODUCT_TYPE[4].Header.RecipeName := '';
   PRODUCT_TYPE[4].Header.RecipeID := 0;
   PRODUCT_TYPE[4].Header."Version" := 0;
   PRODUCT_TYPE[4].Header.LastModified.YEAR := 1970;
   PRODUCT_TYPE[4].Header.LastModified.MONTH := 1;
   PRODUCT_TYPE[4].Header.LastModified.DAY := 1;
   PRODUCT_TYPE[4].Header.LastModified.WEEKDAY := 5;
   PRODUCT_TYPE[4].Header.LastModified.HOUR := 0;
   PRODUCT_TYPE[4].Header.LastModified.MINUTE := 0;
   PRODUCT_TYPE[4].Header.LastModified.SECOND := 0;
   PRODUCT_TYPE[4].Header.LastModified.NANOSECOND := 0;
   PRODUCT_TYPE[4].Header.LastModified := DTL#1970-01-01-00:00:00;
   PRODUCT_TYPE[4].Header.PartType := '';
   PRODUCT_TYPE[4].Header.PartTypeRecordNr := 0;
   PRODUCT_TYPE[4].Process.Timers.Delay_glue_init_start := T#0MS;
   PRODUCT_TYPE[4].Process.Timers.Delay_Medium := T#0MS;
   PRODUCT_TYPE[4].Process.Timers.Delay_Long := T#0MS;
   PRODUCT_TYPE[4].Process.Timers.Cylinder_ActTime := T#0MS;
   PRODUCT_TYPE[4].Process.Limits.RetryLimit := 0;
   PRODUCT_TYPE[4].Process.Press.B1_Program := 0;
   PRODUCT_TYPE[4].Process.Press.B2_Program := 0;
   PRODUCT_TYPE[4].Process.Press.Curve.StartPos_UL := 0.0;
   PRODUCT_TYPE[4].Process.Press.Curve.StartPos_LL := 0.0;
   PRODUCT_TYPE[4].Process.Press.Curve.StartForce_UL := 0.0;
   PRODUCT_TYPE[4].Process.Press.Curve.StartForce_LL := 0.0;
   PRODUCT_TYPE[4].Process.Press.Curve.MiddlePos_UL := 0.0;
   PRODUCT_TYPE[4].Process.Press.Curve.MiddlePos_LL := 0.0;
   PRODUCT_TYPE[4].Process.Press.Curve.MiddleForce_UL := 0.0;
   PRODUCT_TYPE[4].Process.Press.Curve.MiddleForce_LL := 0.0;
   PRODUCT_TYPE[4].Process.Press.Curve.FinalPos_UL := 0.0;
   PRODUCT_TYPE[4].Process.Press.Curve.FinalPos_LL := 0.0;
   PRODUCT_TYPE[4].Process.Press.Curve.FinalForce_UL := 0.0;
   PRODUCT_TYPE[4].Process.Press.Curve.FinalForce_LL := 0.0;
   PRODUCT_TYPE[4].Process.Press.Curve.ProgramNum := 0;
   PRODUCT_TYPE[4].Process.Vision.CGlueShaftIV3_Progs[1] := 16#0000;
   PRODUCT_TYPE[4].Process.Vision.CGlueShaftIV3_Progs[2] := 16#0000;
   PRODUCT_TYPE[4].Process.Vision.CGlueShaftIV3_Progs[3] := 16#0000;
   PRODUCT_TYPE[4].Process.Vision.CGlueShaftIV3_Progs[4] := 16#0000;
   PRODUCT_TYPE[4].Process.Vision.CGlueMagnetIV3_Prog := 16#0000;
   PRODUCT_TYPE[4].Process.Vision.CGlueProgram := 0;
   PRODUCT_TYPE[4]."Tooling Code".A1_Table[1] := '';
   PRODUCT_TYPE[4]."Tooling Code".A1_Table[2] := '';
   PRODUCT_TYPE[4]."Tooling Code".A1_Table[3] := '';
   PRODUCT_TYPE[4]."Tooling Code".A1_Table[4] := '';
   PRODUCT_TYPE[4]."Tooling Code".A1_Table[5] := '';
   PRODUCT_TYPE[4]."Tooling Code".A1_Table[6] := '';
   PRODUCT_TYPE[4]."Tooling Code".A1_Table[7] := '';
   PRODUCT_TYPE[4]."Tooling Code".A1_Table[8] := '';
   PRODUCT_TYPE[4]."Tooling Code".A2_Table[1] := '';
   PRODUCT_TYPE[4]."Tooling Code".A2_Table[2] := '';
   PRODUCT_TYPE[4]."Tooling Code".A2_Table[3] := '';
   PRODUCT_TYPE[4]."Tooling Code".A2_Table[4] := '';
   PRODUCT_TYPE[4]."Tooling Code".A2_Table[5] := '';
   PRODUCT_TYPE[4]."Tooling Code".A2_Table[6] := '';
   PRODUCT_TYPE[4]."Tooling Code".A2_Table[7] := '';
   PRODUCT_TYPE[4]."Tooling Code".A2_Table[8] := '';
   PRODUCT_TYPE[4]."Tooling Code".ROB1_Shaft_Handling_Robot.Gripper."JAW TOOLING LEFT" := '';
   PRODUCT_TYPE[4]."Tooling Code".ROB1_Shaft_Handling_Robot.Gripper."JAW TOOLING RIGHT" := '';
   PRODUCT_TYPE[4]."Tooling Code".ROB1_Shaft_Handling_Robot.Gripper."SHAFT CLAMPING LEFT" := '';
   PRODUCT_TYPE[4]."Tooling Code".ROB1_Shaft_Handling_Robot.Gripper."SHAFT CLAMPING RIGHT" := '';
   PRODUCT_TYPE[4]."Tooling Code".ROB2_Main_Assembly_Robot.Gripper."JAW TOOLING LEFT" := '';
   PRODUCT_TYPE[4]."Tooling Code".ROB2_Main_Assembly_Robot.Gripper."JAW TOOLING RIGHT" := '';
   PRODUCT_TYPE[4]."Tooling Code".ROB2_Main_Assembly_Robot.Gripper."SHAFT CLAMPING LEFT" := '';
   PRODUCT_TYPE[4]."Tooling Code".ROB2_Main_Assembly_Robot.Gripper."SHAFT CLAMPING RIGHT" := '';
   PRODUCT_TYPE[4]."Tooling Code".ROB3_Unloading_Robot.Gripper."JAW TOOLING LEFT" := '';
   PRODUCT_TYPE[4]."Tooling Code".ROB3_Unloading_Robot.Gripper."JAW TOOLING RIGHT" := '';
   PRODUCT_TYPE[4]."Tooling Code".ROB3_Unloading_Robot.Gripper."SHAFT CLAMPING LEFT" := '';
   PRODUCT_TYPE[4]."Tooling Code".ROB3_Unloading_Robot.Gripper."SHAFT CLAMPING RIGHT" := '';
   PRODUCT_TYPE[4]."Tooling Code".A1_Fixtures.A1RingUnloadingFixtureCode := '';
   PRODUCT_TYPE[4]."Tooling Code".A1_Fixtures.E1LoadingNGFixtureCode := '';
   PRODUCT_TYPE[4]."Tooling Code".A1_Fixtures.ShaftScanFixtureCode := '';
   PRODUCT_TYPE[4]."Tooling Code".A1_Fixtures.B1PressFixtureCode := '';
   PRODUCT_TYPE[4]."Tooling Code".A1_Fixtures.CGlueFixtureCode := '';
   PRODUCT_TYPE[4]."Tooling Code".A1_Fixtures.B1PressCylFixtureCode := '';
   PRODUCT_TYPE[4]."Tooling Code".A2_Fixtures.A2RingUnloadingFixtureCode := '';
   PRODUCT_TYPE[4]."Tooling Code".A2_Fixtures.E2UnloadingNGFixtureCode := '';
   PRODUCT_TYPE[4]."Tooling Code".A2_Fixtures.B2PressFixtureCode := '';
   PRODUCT_TYPE[4]."Tooling Code".A2_Fixtures.CGlueNGFixtureCode := '';
   PRODUCT_TYPE[4]."Tooling Code".A2_Fixtures.B2PressCylFixtureCode := '';
   PRODUCT_TYPE[5].Header.RecipeName := '';
   PRODUCT_TYPE[5].Header.RecipeID := 0;
   PRODUCT_TYPE[5].Header."Version" := 0;
   PRODUCT_TYPE[5].Header.LastModified.YEAR := 1970;
   PRODUCT_TYPE[5].Header.LastModified.MONTH := 1;
   PRODUCT_TYPE[5].Header.LastModified.DAY := 1;
   PRODUCT_TYPE[5].Header.LastModified.WEEKDAY := 5;
   PRODUCT_TYPE[5].Header.LastModified.HOUR := 0;
   PRODUCT_TYPE[5].Header.LastModified.MINUTE := 0;
   PRODUCT_TYPE[5].Header.LastModified.SECOND := 0;
   PRODUCT_TYPE[5].Header.LastModified.NANOSECOND := 0;
   PRODUCT_TYPE[5].Header.LastModified := DTL#1970-01-01-00:00:00;
   PRODUCT_TYPE[5].Header.PartType := '';
   PRODUCT_TYPE[5].Header.PartTypeRecordNr := 0;
   PRODUCT_TYPE[5].Process.Timers.Delay_glue_init_start := T#0MS;
   PRODUCT_TYPE[5].Process.Timers.Delay_Medium := T#0MS;
   PRODUCT_TYPE[5].Process.Timers.Delay_Long := T#0MS;
   PRODUCT_TYPE[5].Process.Timers.Cylinder_ActTime := T#0MS;
   PRODUCT_TYPE[5].Process.Limits.RetryLimit := 0;
   PRODUCT_TYPE[5].Process.Press.B1_Program := 0;
   PRODUCT_TYPE[5].Process.Press.B2_Program := 0;
   PRODUCT_TYPE[5].Process.Press.Curve.StartPos_UL := 0.0;
   PRODUCT_TYPE[5].Process.Press.Curve.StartPos_LL := 0.0;
   PRODUCT_TYPE[5].Process.Press.Curve.StartForce_UL := 0.0;
   PRODUCT_TYPE[5].Process.Press.Curve.StartForce_LL := 0.0;
   PRODUCT_TYPE[5].Process.Press.Curve.MiddlePos_UL := 0.0;
   PRODUCT_TYPE[5].Process.Press.Curve.MiddlePos_LL := 0.0;
   PRODUCT_TYPE[5].Process.Press.Curve.MiddleForce_UL := 0.0;
   PRODUCT_TYPE[5].Process.Press.Curve.MiddleForce_LL := 0.0;
   PRODUCT_TYPE[5].Process.Press.Curve.FinalPos_UL := 0.0;
   PRODUCT_TYPE[5].Process.Press.Curve.FinalPos_LL := 0.0;
   PRODUCT_TYPE[5].Process.Press.Curve.FinalForce_UL := 0.0;
   PRODUCT_TYPE[5].Process.Press.Curve.FinalForce_LL := 0.0;
   PRODUCT_TYPE[5].Process.Press.Curve.ProgramNum := 0;
   PRODUCT_TYPE[5].Process.Vision.CGlueShaftIV3_Progs[1] := 16#0000;
   PRODUCT_TYPE[5].Process.Vision.CGlueShaftIV3_Progs[2] := 16#0000;
   PRODUCT_TYPE[5].Process.Vision.CGlueShaftIV3_Progs[3] := 16#0000;
   PRODUCT_TYPE[5].Process.Vision.CGlueShaftIV3_Progs[4] := 16#0000;
   PRODUCT_TYPE[5].Process.Vision.CGlueMagnetIV3_Prog := 16#0000;
   PRODUCT_TYPE[5].Process.Vision.CGlueProgram := 0;
   PRODUCT_TYPE[5]."Tooling Code".A1_Table[1] := '';
   PRODUCT_TYPE[5]."Tooling Code".A1_Table[2] := '';
   PRODUCT_TYPE[5]."Tooling Code".A1_Table[3] := '';
   PRODUCT_TYPE[5]."Tooling Code".A1_Table[4] := '';
   PRODUCT_TYPE[5]."Tooling Code".A1_Table[5] := '';
   PRODUCT_TYPE[5]."Tooling Code".A1_Table[6] := '';
   PRODUCT_TYPE[5]."Tooling Code".A1_Table[7] := '';
   PRODUCT_TYPE[5]."Tooling Code".A1_Table[8] := '';
   PRODUCT_TYPE[5]."Tooling Code".A2_Table[1] := '';
   PRODUCT_TYPE[5]."Tooling Code".A2_Table[2] := '';
   PRODUCT_TYPE[5]."Tooling Code".A2_Table[3] := '';
   PRODUCT_TYPE[5]."Tooling Code".A2_Table[4] := '';
   PRODUCT_TYPE[5]."Tooling Code".A2_Table[5] := '';
   PRODUCT_TYPE[5]."Tooling Code".A2_Table[6] := '';
   PRODUCT_TYPE[5]."Tooling Code".A2_Table[7] := '';
   PRODUCT_TYPE[5]."Tooling Code".A2_Table[8] := '';
   PRODUCT_TYPE[5]."Tooling Code".ROB1_Shaft_Handling_Robot.Gripper."JAW TOOLING LEFT" := '';
   PRODUCT_TYPE[5]."Tooling Code".ROB1_Shaft_Handling_Robot.Gripper."JAW TOOLING RIGHT" := '';
   PRODUCT_TYPE[5]."Tooling Code".ROB1_Shaft_Handling_Robot.Gripper."SHAFT CLAMPING LEFT" := '';
   PRODUCT_TYPE[5]."Tooling Code".ROB1_Shaft_Handling_Robot.Gripper."SHAFT CLAMPING RIGHT" := '';
   PRODUCT_TYPE[5]."Tooling Code".ROB2_Main_Assembly_Robot.Gripper."JAW TOOLING LEFT" := '';
   PRODUCT_TYPE[5]."Tooling Code".ROB2_Main_Assembly_Robot.Gripper."JAW TOOLING RIGHT" := '';
   PRODUCT_TYPE[5]."Tooling Code".ROB2_Main_Assembly_Robot.Gripper."SHAFT CLAMPING LEFT" := '';
   PRODUCT_TYPE[5]."Tooling Code".ROB2_Main_Assembly_Robot.Gripper."SHAFT CLAMPING RIGHT" := '';
   PRODUCT_TYPE[5]."Tooling Code".ROB3_Unloading_Robot.Gripper."JAW TOOLING LEFT" := '';
   PRODUCT_TYPE[5]."Tooling Code".ROB3_Unloading_Robot.Gripper."JAW TOOLING RIGHT" := '';
   PRODUCT_TYPE[5]."Tooling Code".ROB3_Unloading_Robot.Gripper."SHAFT CLAMPING LEFT" := '';
   PRODUCT_TYPE[5]."Tooling Code".ROB3_Unloading_Robot.Gripper."SHAFT CLAMPING RIGHT" := '';
   PRODUCT_TYPE[5]."Tooling Code".A1_Fixtures.A1RingUnloadingFixtureCode := '';
   PRODUCT_TYPE[5]."Tooling Code".A1_Fixtures.E1LoadingNGFixtureCode := '';
   PRODUCT_TYPE[5]."Tooling Code".A1_Fixtures.ShaftScanFixtureCode := '';
   PRODUCT_TYPE[5]."Tooling Code".A1_Fixtures.B1PressFixtureCode := '';
   PRODUCT_TYPE[5]."Tooling Code".A1_Fixtures.CGlueFixtureCode := '';
   PRODUCT_TYPE[5]."Tooling Code".A1_Fixtures.B1PressCylFixtureCode := '';
   PRODUCT_TYPE[5]."Tooling Code".A2_Fixtures.A2RingUnloadingFixtureCode := '';
   PRODUCT_TYPE[5]."Tooling Code".A2_Fixtures.E2UnloadingNGFixtureCode := '';
   PRODUCT_TYPE[5]."Tooling Code".A2_Fixtures.B2PressFixtureCode := '';
   PRODUCT_TYPE[5]."Tooling Code".A2_Fixtures.CGlueNGFixtureCode := '';
   PRODUCT_TYPE[5]."Tooling Code".A2_Fixtures.B2PressCylFixtureCode := '';
   PRODUCT_TYPE[6].Header.RecipeName := '';
   PRODUCT_TYPE[6].Header.RecipeID := 0;
   PRODUCT_TYPE[6].Header."Version" := 0;
   PRODUCT_TYPE[6].Header.LastModified.YEAR := 1970;
   PRODUCT_TYPE[6].Header.LastModified.MONTH := 1;
   PRODUCT_TYPE[6].Header.LastModified.DAY := 1;
   PRODUCT_TYPE[6].Header.LastModified.WEEKDAY := 5;
   PRODUCT_TYPE[6].Header.LastModified.HOUR := 0;
   PRODUCT_TYPE[6].Header.LastModified.MINUTE := 0;
   PRODUCT_TYPE[6].Header.LastModified.SECOND := 0;
   PRODUCT_TYPE[6].Header.LastModified.NANOSECOND := 0;
   PRODUCT_TYPE[6].Header.LastModified := DTL#1970-01-01-00:00:00;
   PRODUCT_TYPE[6].Header.PartType := '';
   PRODUCT_TYPE[6].Header.PartTypeRecordNr := 0;
   PRODUCT_TYPE[6].Process.Timers.Delay_glue_init_start := T#0MS;
   PRODUCT_TYPE[6].Process.Timers.Delay_Medium := T#0MS;
   PRODUCT_TYPE[6].Process.Timers.Delay_Long := T#0MS;
   PRODUCT_TYPE[6].Process.Timers.Cylinder_ActTime := T#0MS;
   PRODUCT_TYPE[6].Process.Limits.RetryLimit := 0;
   PRODUCT_TYPE[6].Process.Press.B1_Program := 0;
   PRODUCT_TYPE[6].Process.Press.B2_Program := 0;
   PRODUCT_TYPE[6].Process.Press.Curve.StartPos_UL := 0.0;
   PRODUCT_TYPE[6].Process.Press.Curve.StartPos_LL := 0.0;
   PRODUCT_TYPE[6].Process.Press.Curve.StartForce_UL := 0.0;
   PRODUCT_TYPE[6].Process.Press.Curve.StartForce_LL := 0.0;
   PRODUCT_TYPE[6].Process.Press.Curve.MiddlePos_UL := 0.0;
   PRODUCT_TYPE[6].Process.Press.Curve.MiddlePos_LL := 0.0;
   PRODUCT_TYPE[6].Process.Press.Curve.MiddleForce_UL := 0.0;
   PRODUCT_TYPE[6].Process.Press.Curve.MiddleForce_LL := 0.0;
   PRODUCT_TYPE[6].Process.Press.Curve.FinalPos_UL := 0.0;
   PRODUCT_TYPE[6].Process.Press.Curve.FinalPos_LL := 0.0;
   PRODUCT_TYPE[6].Process.Press.Curve.FinalForce_UL := 0.0;
   PRODUCT_TYPE[6].Process.Press.Curve.FinalForce_LL := 0.0;
   PRODUCT_TYPE[6].Process.Press.Curve.ProgramNum := 0;
   PRODUCT_TYPE[6].Process.Vision.CGlueShaftIV3_Progs[1] := 16#0000;
   PRODUCT_TYPE[6].Process.Vision.CGlueShaftIV3_Progs[2] := 16#0000;
   PRODUCT_TYPE[6].Process.Vision.CGlueShaftIV3_Progs[3] := 16#0000;
   PRODUCT_TYPE[6].Process.Vision.CGlueShaftIV3_Progs[4] := 16#0000;
   PRODUCT_TYPE[6].Process.Vision.CGlueMagnetIV3_Prog := 16#0000;
   PRODUCT_TYPE[6].Process.Vision.CGlueProgram := 0;
   PRODUCT_TYPE[6]."Tooling Code".A1_Table[1] := '';
   PRODUCT_TYPE[6]."Tooling Code".A1_Table[2] := '';
   PRODUCT_TYPE[6]."Tooling Code".A1_Table[3] := '';
   PRODUCT_TYPE[6]."Tooling Code".A1_Table[4] := '';
   PRODUCT_TYPE[6]."Tooling Code".A1_Table[5] := '';
   PRODUCT_TYPE[6]."Tooling Code".A1_Table[6] := '';
   PRODUCT_TYPE[6]."Tooling Code".A1_Table[7] := '';
   PRODUCT_TYPE[6]."Tooling Code".A1_Table[8] := '';
   PRODUCT_TYPE[6]."Tooling Code".A2_Table[1] := '';
   PRODUCT_TYPE[6]."Tooling Code".A2_Table[2] := '';
   PRODUCT_TYPE[6]."Tooling Code".A2_Table[3] := '';
   PRODUCT_TYPE[6]."Tooling Code".A2_Table[4] := '';
   PRODUCT_TYPE[6]."Tooling Code".A2_Table[5] := '';
   PRODUCT_TYPE[6]."Tooling Code".A2_Table[6] := '';
   PRODUCT_TYPE[6]."Tooling Code".A2_Table[7] := '';
   PRODUCT_TYPE[6]."Tooling Code".A2_Table[8] := '';
   PRODUCT_TYPE[6]."Tooling Code".ROB1_Shaft_Handling_Robot.Gripper."JAW TOOLING LEFT" := '';
   PRODUCT_TYPE[6]."Tooling Code".ROB1_Shaft_Handling_Robot.Gripper."JAW TOOLING RIGHT" := '';
   PRODUCT_TYPE[6]."Tooling Code".ROB1_Shaft_Handling_Robot.Gripper."SHAFT CLAMPING LEFT" := '';
   PRODUCT_TYPE[6]."Tooling Code".ROB1_Shaft_Handling_Robot.Gripper."SHAFT CLAMPING RIGHT" := '';
   PRODUCT_TYPE[6]."Tooling Code".ROB2_Main_Assembly_Robot.Gripper."JAW TOOLING LEFT" := '';
   PRODUCT_TYPE[6]."Tooling Code".ROB2_Main_Assembly_Robot.Gripper."JAW TOOLING RIGHT" := '';
   PRODUCT_TYPE[6]."Tooling Code".ROB2_Main_Assembly_Robot.Gripper."SHAFT CLAMPING LEFT" := '';
   PRODUCT_TYPE[6]."Tooling Code".ROB2_Main_Assembly_Robot.Gripper."SHAFT CLAMPING RIGHT" := '';
   PRODUCT_TYPE[6]."Tooling Code".ROB3_Unloading_Robot.Gripper."JAW TOOLING LEFT" := '';
   PRODUCT_TYPE[6]."Tooling Code".ROB3_Unloading_Robot.Gripper."JAW TOOLING RIGHT" := '';
   PRODUCT_TYPE[6]."Tooling Code".ROB3_Unloading_Robot.Gripper."SHAFT CLAMPING LEFT" := '';
   PRODUCT_TYPE[6]."Tooling Code".ROB3_Unloading_Robot.Gripper."SHAFT CLAMPING RIGHT" := '';
   PRODUCT_TYPE[6]."Tooling Code".A1_Fixtures.A1RingUnloadingFixtureCode := '';
   PRODUCT_TYPE[6]."Tooling Code".A1_Fixtures.E1LoadingNGFixtureCode := '';
   PRODUCT_TYPE[6]."Tooling Code".A1_Fixtures.ShaftScanFixtureCode := '';
   PRODUCT_TYPE[6]."Tooling Code".A1_Fixtures.B1PressFixtureCode := '';
   PRODUCT_TYPE[6]."Tooling Code".A1_Fixtures.CGlueFixtureCode := '';
   PRODUCT_TYPE[6]."Tooling Code".A1_Fixtures.B1PressCylFixtureCode := '';
   PRODUCT_TYPE[6]."Tooling Code".A2_Fixtures.A2RingUnloadingFixtureCode := '';
   PRODUCT_TYPE[6]."Tooling Code".A2_Fixtures.E2UnloadingNGFixtureCode := '';
   PRODUCT_TYPE[6]."Tooling Code".A2_Fixtures.B2PressFixtureCode := '';
   PRODUCT_TYPE[6]."Tooling Code".A2_Fixtures.CGlueNGFixtureCode := '';
   PRODUCT_TYPE[6]."Tooling Code".A2_Fixtures.B2PressCylFixtureCode := '';
   PRODUCT_TYPE[7].Header.RecipeName := '';
   PRODUCT_TYPE[7].Header.RecipeID := 0;
   PRODUCT_TYPE[7].Header."Version" := 0;
   PRODUCT_TYPE[7].Header.LastModified.YEAR := 1970;
   PRODUCT_TYPE[7].Header.LastModified.MONTH := 1;
   PRODUCT_TYPE[7].Header.LastModified.DAY := 1;
   PRODUCT_TYPE[7].Header.LastModified.WEEKDAY := 5;
   PRODUCT_TYPE[7].Header.LastModified.HOUR := 0;
   PRODUCT_TYPE[7].Header.LastModified.MINUTE := 0;
   PRODUCT_TYPE[7].Header.LastModified.SECOND := 0;
   PRODUCT_TYPE[7].Header.LastModified.NANOSECOND := 0;
   PRODUCT_TYPE[7].Header.LastModified := DTL#1970-01-01-00:00:00;
   PRODUCT_TYPE[7].Header.PartType := '';
   PRODUCT_TYPE[7].Header.PartTypeRecordNr := 0;
   PRODUCT_TYPE[7].Process.Timers.Delay_glue_init_start := T#0MS;
   PRODUCT_TYPE[7].Process.Timers.Delay_Medium := T#0MS;
   PRODUCT_TYPE[7].Process.Timers.Delay_Long := T#0MS;
   PRODUCT_TYPE[7].Process.Timers.Cylinder_ActTime := T#0MS;
   PRODUCT_TYPE[7].Process.Limits.RetryLimit := 0;
   PRODUCT_TYPE[7].Process.Press.B1_Program := 0;
   PRODUCT_TYPE[7].Process.Press.B2_Program := 0;
   PRODUCT_TYPE[7].Process.Press.Curve.StartPos_UL := 0.0;
   PRODUCT_TYPE[7].Process.Press.Curve.StartPos_LL := 0.0;
   PRODUCT_TYPE[7].Process.Press.Curve.StartForce_UL := 0.0;
   PRODUCT_TYPE[7].Process.Press.Curve.StartForce_LL := 0.0;
   PRODUCT_TYPE[7].Process.Press.Curve.MiddlePos_UL := 0.0;
   PRODUCT_TYPE[7].Process.Press.Curve.MiddlePos_LL := 0.0;
   PRODUCT_TYPE[7].Process.Press.Curve.MiddleForce_UL := 0.0;
   PRODUCT_TYPE[7].Process.Press.Curve.MiddleForce_LL := 0.0;
   PRODUCT_TYPE[7].Process.Press.Curve.FinalPos_UL := 0.0;
   PRODUCT_TYPE[7].Process.Press.Curve.FinalPos_LL := 0.0;
   PRODUCT_TYPE[7].Process.Press.Curve.FinalForce_UL := 0.0;
   PRODUCT_TYPE[7].Process.Press.Curve.FinalForce_LL := 0.0;
   PRODUCT_TYPE[7].Process.Press.Curve.ProgramNum := 0;
   PRODUCT_TYPE[7].Process.Vision.CGlueShaftIV3_Progs[1] := 16#0000;
   PRODUCT_TYPE[7].Process.Vision.CGlueShaftIV3_Progs[2] := 16#0000;
   PRODUCT_TYPE[7].Process.Vision.CGlueShaftIV3_Progs[3] := 16#0000;
   PRODUCT_TYPE[7].Process.Vision.CGlueShaftIV3_Progs[4] := 16#0000;
   PRODUCT_TYPE[7].Process.Vision.CGlueMagnetIV3_Prog := 16#0000;
   PRODUCT_TYPE[7].Process.Vision.CGlueProgram := 0;
   PRODUCT_TYPE[7]."Tooling Code".A1_Table[1] := '';
   PRODUCT_TYPE[7]."Tooling Code".A1_Table[2] := '';
   PRODUCT_TYPE[7]."Tooling Code".A1_Table[3] := '';
   PRODUCT_TYPE[7]."Tooling Code".A1_Table[4] := '';
   PRODUCT_TYPE[7]."Tooling Code".A1_Table[5] := '';
   PRODUCT_TYPE[7]."Tooling Code".A1_Table[6] := '';
   PRODUCT_TYPE[7]."Tooling Code".A1_Table[7] := '';
   PRODUCT_TYPE[7]."Tooling Code".A1_Table[8] := '';
   PRODUCT_TYPE[7]."Tooling Code".A2_Table[1] := '';
   PRODUCT_TYPE[7]."Tooling Code".A2_Table[2] := '';
   PRODUCT_TYPE[7]."Tooling Code".A2_Table[3] := '';
   PRODUCT_TYPE[7]."Tooling Code".A2_Table[4] := '';
   PRODUCT_TYPE[7]."Tooling Code".A2_Table[5] := '';
   PRODUCT_TYPE[7]."Tooling Code".A2_Table[6] := '';
   PRODUCT_TYPE[7]."Tooling Code".A2_Table[7] := '';
   PRODUCT_TYPE[7]."Tooling Code".A2_Table[8] := '';
   PRODUCT_TYPE[7]."Tooling Code".ROB1_Shaft_Handling_Robot.Gripper."JAW TOOLING LEFT" := '';
   PRODUCT_TYPE[7]."Tooling Code".ROB1_Shaft_Handling_Robot.Gripper."JAW TOOLING RIGHT" := '';
   PRODUCT_TYPE[7]."Tooling Code".ROB1_Shaft_Handling_Robot.Gripper."SHAFT CLAMPING LEFT" := '';
   PRODUCT_TYPE[7]."Tooling Code".ROB1_Shaft_Handling_Robot.Gripper."SHAFT CLAMPING RIGHT" := '';
   PRODUCT_TYPE[7]."Tooling Code".ROB2_Main_Assembly_Robot.Gripper."JAW TOOLING LEFT" := '';
   PRODUCT_TYPE[7]."Tooling Code".ROB2_Main_Assembly_Robot.Gripper."JAW TOOLING RIGHT" := '';
   PRODUCT_TYPE[7]."Tooling Code".ROB2_Main_Assembly_Robot.Gripper."SHAFT CLAMPING LEFT" := '';
   PRODUCT_TYPE[7]."Tooling Code".ROB2_Main_Assembly_Robot.Gripper."SHAFT CLAMPING RIGHT" := '';
   PRODUCT_TYPE[7]."Tooling Code".ROB3_Unloading_Robot.Gripper."JAW TOOLING LEFT" := '';
   PRODUCT_TYPE[7]."Tooling Code".ROB3_Unloading_Robot.Gripper."JAW TOOLING RIGHT" := '';
   PRODUCT_TYPE[7]."Tooling Code".ROB3_Unloading_Robot.Gripper."SHAFT CLAMPING LEFT" := '';
   PRODUCT_TYPE[7]."Tooling Code".ROB3_Unloading_Robot.Gripper."SHAFT CLAMPING RIGHT" := '';
   PRODUCT_TYPE[7]."Tooling Code".A1_Fixtures.A1RingUnloadingFixtureCode := '';
   PRODUCT_TYPE[7]."Tooling Code".A1_Fixtures.E1LoadingNGFixtureCode := '';
   PRODUCT_TYPE[7]."Tooling Code".A1_Fixtures.ShaftScanFixtureCode := '';
   PRODUCT_TYPE[7]."Tooling Code".A1_Fixtures.B1PressFixtureCode := '';
   PRODUCT_TYPE[7]."Tooling Code".A1_Fixtures.CGlueFixtureCode := '';
   PRODUCT_TYPE[7]."Tooling Code".A1_Fixtures.B1PressCylFixtureCode := '';
   PRODUCT_TYPE[7]."Tooling Code".A2_Fixtures.A2RingUnloadingFixtureCode := '';
   PRODUCT_TYPE[7]."Tooling Code".A2_Fixtures.E2UnloadingNGFixtureCode := '';
   PRODUCT_TYPE[7]."Tooling Code".A2_Fixtures.B2PressFixtureCode := '';
   PRODUCT_TYPE[7]."Tooling Code".A2_Fixtures.CGlueNGFixtureCode := '';
   PRODUCT_TYPE[7]."Tooling Code".A2_Fixtures.B2PressCylFixtureCode := '';
   PRODUCT_TYPE[8].Header.RecipeName := '';
   PRODUCT_TYPE[8].Header.RecipeID := 0;
   PRODUCT_TYPE[8].Header."Version" := 0;
   PRODUCT_TYPE[8].Header.LastModified.YEAR := 1970;
   PRODUCT_TYPE[8].Header.LastModified.MONTH := 1;
   PRODUCT_TYPE[8].Header.LastModified.DAY := 1;
   PRODUCT_TYPE[8].Header.LastModified.WEEKDAY := 5;
   PRODUCT_TYPE[8].Header.LastModified.HOUR := 0;
   PRODUCT_TYPE[8].Header.LastModified.MINUTE := 0;
   PRODUCT_TYPE[8].Header.LastModified.SECOND := 0;
   PRODUCT_TYPE[8].Header.LastModified.NANOSECOND := 0;
   PRODUCT_TYPE[8].Header.LastModified := DTL#1970-01-01-00:00:00;
   PRODUCT_TYPE[8].Header.PartType := '';
   PRODUCT_TYPE[8].Header.PartTypeRecordNr := 0;
   PRODUCT_TYPE[8].Process.Timers.Delay_glue_init_start := T#0MS;
   PRODUCT_TYPE[8].Process.Timers.Delay_Medium := T#0MS;
   PRODUCT_TYPE[8].Process.Timers.Delay_Long := T#0MS;
   PRODUCT_TYPE[8].Process.Timers.Cylinder_ActTime := T#0MS;
   PRODUCT_TYPE[8].Process.Limits.RetryLimit := 0;
   PRODUCT_TYPE[8].Process.Press.B1_Program := 0;
   PRODUCT_TYPE[8].Process.Press.B2_Program := 0;
   PRODUCT_TYPE[8].Process.Press.Curve.StartPos_UL := 0.0;
   PRODUCT_TYPE[8].Process.Press.Curve.StartPos_LL := 0.0;
   PRODUCT_TYPE[8].Process.Press.Curve.StartForce_UL := 0.0;
   PRODUCT_TYPE[8].Process.Press.Curve.StartForce_LL := 0.0;
   PRODUCT_TYPE[8].Process.Press.Curve.MiddlePos_UL := 0.0;
   PRODUCT_TYPE[8].Process.Press.Curve.MiddlePos_LL := 0.0;
   PRODUCT_TYPE[8].Process.Press.Curve.MiddleForce_UL := 0.0;
   PRODUCT_TYPE[8].Process.Press.Curve.MiddleForce_LL := 0.0;
   PRODUCT_TYPE[8].Process.Press.Curve.FinalPos_UL := 0.0;
   PRODUCT_TYPE[8].Process.Press.Curve.FinalPos_LL := 0.0;
   PRODUCT_TYPE[8].Process.Press.Curve.FinalForce_UL := 0.0;
   PRODUCT_TYPE[8].Process.Press.Curve.FinalForce_LL := 0.0;
   PRODUCT_TYPE[8].Process.Press.Curve.ProgramNum := 0;
   PRODUCT_TYPE[8].Process.Vision.CGlueShaftIV3_Progs[1] := 16#0000;
   PRODUCT_TYPE[8].Process.Vision.CGlueShaftIV3_Progs[2] := 16#0000;
   PRODUCT_TYPE[8].Process.Vision.CGlueShaftIV3_Progs[3] := 16#0000;
   PRODUCT_TYPE[8].Process.Vision.CGlueShaftIV3_Progs[4] := 16#0000;
   PRODUCT_TYPE[8].Process.Vision.CGlueMagnetIV3_Prog := 16#0000;
   PRODUCT_TYPE[8].Process.Vision.CGlueProgram := 0;
   PRODUCT_TYPE[8]."Tooling Code".A1_Table[1] := '';
   PRODUCT_TYPE[8]."Tooling Code".A1_Table[2] := '';
   PRODUCT_TYPE[8]."Tooling Code".A1_Table[3] := '';
   PRODUCT_TYPE[8]."Tooling Code".A1_Table[4] := '';
   PRODUCT_TYPE[8]."Tooling Code".A1_Table[5] := '';
   PRODUCT_TYPE[8]."Tooling Code".A1_Table[6] := '';
   PRODUCT_TYPE[8]."Tooling Code".A1_Table[7] := '';
   PRODUCT_TYPE[8]."Tooling Code".A1_Table[8] := '';
   PRODUCT_TYPE[8]."Tooling Code".A2_Table[1] := '';
   PRODUCT_TYPE[8]."Tooling Code".A2_Table[2] := '';
   PRODUCT_TYPE[8]."Tooling Code".A2_Table[3] := '';
   PRODUCT_TYPE[8]."Tooling Code".A2_Table[4] := '';
   PRODUCT_TYPE[8]."Tooling Code".A2_Table[5] := '';
   PRODUCT_TYPE[8]."Tooling Code".A2_Table[6] := '';
   PRODUCT_TYPE[8]."Tooling Code".A2_Table[7] := '';
   PRODUCT_TYPE[8]."Tooling Code".A2_Table[8] := '';
   PRODUCT_TYPE[8]."Tooling Code".ROB1_Shaft_Handling_Robot.Gripper."JAW TOOLING LEFT" := '';
   PRODUCT_TYPE[8]."Tooling Code".ROB1_Shaft_Handling_Robot.Gripper."JAW TOOLING RIGHT" := '';
   PRODUCT_TYPE[8]."Tooling Code".ROB1_Shaft_Handling_Robot.Gripper."SHAFT CLAMPING LEFT" := '';
   PRODUCT_TYPE[8]."Tooling Code".ROB1_Shaft_Handling_Robot.Gripper."SHAFT CLAMPING RIGHT" := '';
   PRODUCT_TYPE[8]."Tooling Code".ROB2_Main_Assembly_Robot.Gripper."JAW TOOLING LEFT" := '';
   PRODUCT_TYPE[8]."Tooling Code".ROB2_Main_Assembly_Robot.Gripper."JAW TOOLING RIGHT" := '';
   PRODUCT_TYPE[8]."Tooling Code".ROB2_Main_Assembly_Robot.Gripper."SHAFT CLAMPING LEFT" := '';
   PRODUCT_TYPE[8]."Tooling Code".ROB2_Main_Assembly_Robot.Gripper."SHAFT CLAMPING RIGHT" := '';
   PRODUCT_TYPE[8]."Tooling Code".ROB3_Unloading_Robot.Gripper."JAW TOOLING LEFT" := '';
   PRODUCT_TYPE[8]."Tooling Code".ROB3_Unloading_Robot.Gripper."JAW TOOLING RIGHT" := '';
   PRODUCT_TYPE[8]."Tooling Code".ROB3_Unloading_Robot.Gripper."SHAFT CLAMPING LEFT" := '';
   PRODUCT_TYPE[8]."Tooling Code".ROB3_Unloading_Robot.Gripper."SHAFT CLAMPING RIGHT" := '';
   PRODUCT_TYPE[8]."Tooling Code".A1_Fixtures.A1RingUnloadingFixtureCode := '';
   PRODUCT_TYPE[8]."Tooling Code".A1_Fixtures.E1LoadingNGFixtureCode := '';
   PRODUCT_TYPE[8]."Tooling Code".A1_Fixtures.ShaftScanFixtureCode := '';
   PRODUCT_TYPE[8]."Tooling Code".A1_Fixtures.B1PressFixtureCode := '';
   PRODUCT_TYPE[8]."Tooling Code".A1_Fixtures.CGlueFixtureCode := '';
   PRODUCT_TYPE[8]."Tooling Code".A1_Fixtures.B1PressCylFixtureCode := '';
   PRODUCT_TYPE[8]."Tooling Code".A2_Fixtures.A2RingUnloadingFixtureCode := '';
   PRODUCT_TYPE[8]."Tooling Code".A2_Fixtures.E2UnloadingNGFixtureCode := '';
   PRODUCT_TYPE[8]."Tooling Code".A2_Fixtures.B2PressFixtureCode := '';
   PRODUCT_TYPE[8]."Tooling Code".A2_Fixtures.CGlueNGFixtureCode := '';
   PRODUCT_TYPE[8]."Tooling Code".A2_Fixtures.B2PressCylFixtureCode := '';
   PRODUCT_TYPE[9].Header.RecipeName := '';
   PRODUCT_TYPE[9].Header.RecipeID := 0;
   PRODUCT_TYPE[9].Header."Version" := 0;
   PRODUCT_TYPE[9].Header.LastModified.YEAR := 1970;
   PRODUCT_TYPE[9].Header.LastModified.MONTH := 1;
   PRODUCT_TYPE[9].Header.LastModified.DAY := 1;
   PRODUCT_TYPE[9].Header.LastModified.WEEKDAY := 5;
   PRODUCT_TYPE[9].Header.LastModified.HOUR := 0;
   PRODUCT_TYPE[9].Header.LastModified.MINUTE := 0;
   PRODUCT_TYPE[9].Header.LastModified.SECOND := 0;
   PRODUCT_TYPE[9].Header.LastModified.NANOSECOND := 0;
   PRODUCT_TYPE[9].Header.LastModified := DTL#1970-01-01-00:00:00;
   PRODUCT_TYPE[9].Header.PartType := '';
   PRODUCT_TYPE[9].Header.PartTypeRecordNr := 0;
   PRODUCT_TYPE[9].Process.Timers.Delay_glue_init_start := T#0MS;
   PRODUCT_TYPE[9].Process.Timers.Delay_Medium := T#0MS;
   PRODUCT_TYPE[9].Process.Timers.Delay_Long := T#0MS;
   PRODUCT_TYPE[9].Process.Timers.Cylinder_ActTime := T#0MS;
   PRODUCT_TYPE[9].Process.Limits.RetryLimit := 0;
   PRODUCT_TYPE[9].Process.Press.B1_Program := 0;
   PRODUCT_TYPE[9].Process.Press.B2_Program := 0;
   PRODUCT_TYPE[9].Process.Press.Curve.StartPos_UL := 0.0;
   PRODUCT_TYPE[9].Process.Press.Curve.StartPos_LL := 0.0;
   PRODUCT_TYPE[9].Process.Press.Curve.StartForce_UL := 0.0;
   PRODUCT_TYPE[9].Process.Press.Curve.StartForce_LL := 0.0;
   PRODUCT_TYPE[9].Process.Press.Curve.MiddlePos_UL := 0.0;
   PRODUCT_TYPE[9].Process.Press.Curve.MiddlePos_LL := 0.0;
   PRODUCT_TYPE[9].Process.Press.Curve.MiddleForce_UL := 0.0;
   PRODUCT_TYPE[9].Process.Press.Curve.MiddleForce_LL := 0.0;
   PRODUCT_TYPE[9].Process.Press.Curve.FinalPos_UL := 0.0;
   PRODUCT_TYPE[9].Process.Press.Curve.FinalPos_LL := 0.0;
   PRODUCT_TYPE[9].Process.Press.Curve.FinalForce_UL := 0.0;
   PRODUCT_TYPE[9].Process.Press.Curve.FinalForce_LL := 0.0;
   PRODUCT_TYPE[9].Process.Press.Curve.ProgramNum := 0;
   PRODUCT_TYPE[9].Process.Vision.CGlueShaftIV3_Progs[1] := 16#0000;
   PRODUCT_TYPE[9].Process.Vision.CGlueShaftIV3_Progs[2] := 16#0000;
   PRODUCT_TYPE[9].Process.Vision.CGlueShaftIV3_Progs[3] := 16#0000;
   PRODUCT_TYPE[9].Process.Vision.CGlueShaftIV3_Progs[4] := 16#0000;
   PRODUCT_TYPE[9].Process.Vision.CGlueMagnetIV3_Prog := 16#0000;
   PRODUCT_TYPE[9].Process.Vision.CGlueProgram := 0;
   PRODUCT_TYPE[9]."Tooling Code".A1_Table[1] := '';
   PRODUCT_TYPE[9]."Tooling Code".A1_Table[2] := '';
   PRODUCT_TYPE[9]."Tooling Code".A1_Table[3] := '';
   PRODUCT_TYPE[9]."Tooling Code".A1_Table[4] := '';
   PRODUCT_TYPE[9]."Tooling Code".A1_Table[5] := '';
   PRODUCT_TYPE[9]."Tooling Code".A1_Table[6] := '';
   PRODUCT_TYPE[9]."Tooling Code".A1_Table[7] := '';
   PRODUCT_TYPE[9]."Tooling Code".A1_Table[8] := '';
   PRODUCT_TYPE[9]."Tooling Code".A2_Table[1] := '';
   PRODUCT_TYPE[9]."Tooling Code".A2_Table[2] := '';
   PRODUCT_TYPE[9]."Tooling Code".A2_Table[3] := '';
   PRODUCT_TYPE[9]."Tooling Code".A2_Table[4] := '';
   PRODUCT_TYPE[9]."Tooling Code".A2_Table[5] := '';
   PRODUCT_TYPE[9]."Tooling Code".A2_Table[6] := '';
   PRODUCT_TYPE[9]."Tooling Code".A2_Table[7] := '';
   PRODUCT_TYPE[9]."Tooling Code".A2_Table[8] := '';
   PRODUCT_TYPE[9]."Tooling Code".ROB1_Shaft_Handling_Robot.Gripper."JAW TOOLING LEFT" := '';
   PRODUCT_TYPE[9]."Tooling Code".ROB1_Shaft_Handling_Robot.Gripper."JAW TOOLING RIGHT" := '';
   PRODUCT_TYPE[9]."Tooling Code".ROB1_Shaft_Handling_Robot.Gripper."SHAFT CLAMPING LEFT" := '';
   PRODUCT_TYPE[9]."Tooling Code".ROB1_Shaft_Handling_Robot.Gripper."SHAFT CLAMPING RIGHT" := '';
   PRODUCT_TYPE[9]."Tooling Code".ROB2_Main_Assembly_Robot.Gripper."JAW TOOLING LEFT" := '';
   PRODUCT_TYPE[9]."Tooling Code".ROB2_Main_Assembly_Robot.Gripper."JAW TOOLING RIGHT" := '';
   PRODUCT_TYPE[9]."Tooling Code".ROB2_Main_Assembly_Robot.Gripper."SHAFT CLAMPING LEFT" := '';
   PRODUCT_TYPE[9]."Tooling Code".ROB2_Main_Assembly_Robot.Gripper."SHAFT CLAMPING RIGHT" := '';
   PRODUCT_TYPE[9]."Tooling Code".ROB3_Unloading_Robot.Gripper."JAW TOOLING LEFT" := '';
   PRODUCT_TYPE[9]."Tooling Code".ROB3_Unloading_Robot.Gripper."JAW TOOLING RIGHT" := '';
   PRODUCT_TYPE[9]."Tooling Code".ROB3_Unloading_Robot.Gripper."SHAFT CLAMPING LEFT" := '';
   PRODUCT_TYPE[9]."Tooling Code".ROB3_Unloading_Robot.Gripper."SHAFT CLAMPING RIGHT" := '';
   PRODUCT_TYPE[9]."Tooling Code".A1_Fixtures.A1RingUnloadingFixtureCode := '';
   PRODUCT_TYPE[9]."Tooling Code".A1_Fixtures.E1LoadingNGFixtureCode := '';
   PRODUCT_TYPE[9]."Tooling Code".A1_Fixtures.ShaftScanFixtureCode := '';
   PRODUCT_TYPE[9]."Tooling Code".A1_Fixtures.B1PressFixtureCode := '';
   PRODUCT_TYPE[9]."Tooling Code".A1_Fixtures.CGlueFixtureCode := '';
   PRODUCT_TYPE[9]."Tooling Code".A1_Fixtures.B1PressCylFixtureCode := '';
   PRODUCT_TYPE[9]."Tooling Code".A2_Fixtures.A2RingUnloadingFixtureCode := '';
   PRODUCT_TYPE[9]."Tooling Code".A2_Fixtures.E2UnloadingNGFixtureCode := '';
   PRODUCT_TYPE[9]."Tooling Code".A2_Fixtures.B2PressFixtureCode := '';
   PRODUCT_TYPE[9]."Tooling Code".A2_Fixtures.CGlueNGFixtureCode := '';
   PRODUCT_TYPE[9]."Tooling Code".A2_Fixtures.B2PressCylFixtureCode := '';
   PRODUCT_TYPE[10].Header.RecipeName := 'produkt 1';
   PRODUCT_TYPE[10].Header.RecipeID := 1;
   PRODUCT_TYPE[10].Header."Version" := 1;
   PRODUCT_TYPE[10].Header.LastModified.YEAR := 2026;
   PRODUCT_TYPE[10].Header.LastModified.MONTH := 1;
   PRODUCT_TYPE[10].Header.LastModified.DAY := 17;
   PRODUCT_TYPE[10].Header.LastModified.WEEKDAY := 7;
   PRODUCT_TYPE[10].Header.LastModified.HOUR := 4;
   PRODUCT_TYPE[10].Header.LastModified.MINUTE := 23;
   PRODUCT_TYPE[10].Header.LastModified.SECOND := 27;
   PRODUCT_TYPE[10].Header.LastModified.NANOSECOND := 501000000;
   PRODUCT_TYPE[10].Header.LastModified := DTL#2026-01-17-04:23:27.501;
   PRODUCT_TYPE[10].Header.PartType := 'additional  name';
   PRODUCT_TYPE[10].Header.PartTypeRecordNr := 0;
   PRODUCT_TYPE[10].Process.Timers.Delay_glue_init_start := T#2S;
   PRODUCT_TYPE[10].Process.Timers.Delay_Medium := T#600MS;
   PRODUCT_TYPE[10].Process.Timers.Delay_Long := T#2S;
   PRODUCT_TYPE[10].Process.Timers.Cylinder_ActTime := T#6S;
   PRODUCT_TYPE[10].Process.Limits.RetryLimit := 3;
   PRODUCT_TYPE[10].Process.Press.B1_Program := 1;
   PRODUCT_TYPE[10].Process.Press.B2_Program := 1;
   PRODUCT_TYPE[10].Process.Press.Curve.StartPos_UL := 0.0;
   PRODUCT_TYPE[10].Process.Press.Curve.StartPos_LL := 0.0;
   PRODUCT_TYPE[10].Process.Press.Curve.StartForce_UL := 0.0;
   PRODUCT_TYPE[10].Process.Press.Curve.StartForce_LL := 0.0;
   PRODUCT_TYPE[10].Process.Press.Curve.MiddlePos_UL := 0.0;
   PRODUCT_TYPE[10].Process.Press.Curve.MiddlePos_LL := 0.0;
   PRODUCT_TYPE[10].Process.Press.Curve.MiddleForce_UL := 0.0;
   PRODUCT_TYPE[10].Process.Press.Curve.MiddleForce_LL := 0.0;
   PRODUCT_TYPE[10].Process.Press.Curve.FinalPos_UL := 0.0;
   PRODUCT_TYPE[10].Process.Press.Curve.FinalPos_LL := 0.0;
   PRODUCT_TYPE[10].Process.Press.Curve.FinalForce_UL := 0.0;
   PRODUCT_TYPE[10].Process.Press.Curve.FinalForce_LL := 0.0;
   PRODUCT_TYPE[10].Process.Press.Curve.ProgramNum := 0;
   PRODUCT_TYPE[10].Process.Vision.CGlueShaftIV3_Progs[1] := 16#0001;
   PRODUCT_TYPE[10].Process.Vision.CGlueShaftIV3_Progs[2] := 16#0002;
   PRODUCT_TYPE[10].Process.Vision.CGlueShaftIV3_Progs[3] := 16#0003;
   PRODUCT_TYPE[10].Process.Vision.CGlueShaftIV3_Progs[4] := 16#0004;
   PRODUCT_TYPE[10].Process.Vision.CGlueMagnetIV3_Prog := 16#0001;
   PRODUCT_TYPE[10].Process.Vision.CGlueProgram := 1;
   PRODUCT_TYPE[10]."Tooling Code".A1_Table[1] := 'SZ23055-OP010-E-Compressor-ring1 Loading tooling-1';
   PRODUCT_TYPE[10]."Tooling Code".A1_Table[2] := 'SZ23055-OP010-E-Compressor-ring1 Loading tooling-2';
   PRODUCT_TYPE[10]."Tooling Code".A1_Table[3] := 'SZ23055-OP010-E-Compressor-ring1 Loading tooling-3';
   PRODUCT_TYPE[10]."Tooling Code".A1_Table[4] := 'SZ23055-OP010-E-Compressor-ring1 Loading tooling-4';
   PRODUCT_TYPE[10]."Tooling Code".A1_Table[5] := 'SZ23055-OP010-E-Compressor-ring1 Loading tooling-5';
   PRODUCT_TYPE[10]."Tooling Code".A1_Table[6] := 'SZ23055-OP010-E-Compressor-ring1 Loading tooling-6';
   PRODUCT_TYPE[10]."Tooling Code".A1_Table[7] := 'SZ23055-OP010-E-Compressor-ring1 Loading tooling-7';
   PRODUCT_TYPE[10]."Tooling Code".A1_Table[8] := 'SZ23055-OP010-E-Compressor-ring1 Loading tooling-8';
   PRODUCT_TYPE[10]."Tooling Code".A2_Table[1] := 'SZ23055-OP010-E-Compresspr-ring1 cutting tool';
   PRODUCT_TYPE[10]."Tooling Code".A2_Table[2] := 'SZ23055-OP010-E-Compressor-Left NG tooling-1';
   PRODUCT_TYPE[10]."Tooling Code".A2_Table[3] := 'SZ23055-OP010-E-Compressor-shaft Rotating scanning tooling-1';
   PRODUCT_TYPE[10]."Tooling Code".A2_Table[4] := 'SZ23055-OP010-E-Compressor-ring1 Below Positioning fixture -1';
   PRODUCT_TYPE[10]."Tooling Code".A2_Table[5] := 'SZ23055-OP010-E-Compressor-Point adhesive tooling-1';
   PRODUCT_TYPE[10]."Tooling Code".A2_Table[6] := 'SZ23055-OP010-E-Compressor-ring1 Upper pressing fixture-1';
   PRODUCT_TYPE[10]."Tooling Code".A2_Table[7] := 'SZ23055-OP010-E-Compresspr-ring2 cutting tool';
   PRODUCT_TYPE[10]."Tooling Code".A2_Table[8] := 'SZ23055-OP010-E-Compressor-Right NG tooling-1';
   PRODUCT_TYPE[10]."Tooling Code".ROB1_Shaft_Handling_Robot.Gripper."JAW TOOLING LEFT" := 'SZ23055-OP010-E-Compressor-robot1 ring1 Left clamping jaw tooling-1';
   PRODUCT_TYPE[10]."Tooling Code".ROB1_Shaft_Handling_Robot.Gripper."JAW TOOLING RIGHT" := 'SZ23055-OP010-E-Compressor-robot1 ring1 Right clamping jaw tooling-2';
   PRODUCT_TYPE[10]."Tooling Code".ROB1_Shaft_Handling_Robot.Gripper."SHAFT CLAMPING LEFT" := 'SZ23055-OP010-E-Compressor-robot1 shaft Left clamping jaw tooling-1';
   PRODUCT_TYPE[10]."Tooling Code".ROB1_Shaft_Handling_Robot.Gripper."SHAFT CLAMPING RIGHT" := 'SZ23055-OP010-E-Compressor-robot1 shaft Right clamping jaw tooling-2';
   PRODUCT_TYPE[10]."Tooling Code".ROB2_Main_Assembly_Robot.Gripper."JAW TOOLING LEFT" := 'SZ23055-OP010-E-Compressor-robot2 shaft Right clamping jaw tooling-2';
   PRODUCT_TYPE[10]."Tooling Code".ROB2_Main_Assembly_Robot.Gripper."JAW TOOLING RIGHT" := 'SZ23055-OP010-E-Compressor-robot2 shaft Left clamping jaw tooling-1';
   PRODUCT_TYPE[10]."Tooling Code".ROB2_Main_Assembly_Robot.Gripper."SHAFT CLAMPING LEFT" := 'SZ23055-OP010-E-Compressor-robot2 magnet Right clamping jaw tooling-2';
   PRODUCT_TYPE[10]."Tooling Code".ROB2_Main_Assembly_Robot.Gripper."SHAFT CLAMPING RIGHT" := 'SZ23055-OP010-E-Compressor-robot2 magnet Right clamping jaw tooling-2';
   PRODUCT_TYPE[10]."Tooling Code".ROB3_Unloading_Robot.Gripper."JAW TOOLING LEFT" := 'SZ23055-OP010-E-Compressor-robot3 ring2 Right clamping jaw tooling-2';
   PRODUCT_TYPE[10]."Tooling Code".ROB3_Unloading_Robot.Gripper."JAW TOOLING RIGHT" := 'SZ23055-OP010-E-Compressor-robot3 ring2 Left clamping jaw tooling-1';
   PRODUCT_TYPE[10]."Tooling Code".ROB3_Unloading_Robot.Gripper."SHAFT CLAMPING LEFT" := 'SZ23055-OP010-E-Compressor-robot3 shaft Left clamping jaw tooling-1';
   PRODUCT_TYPE[10]."Tooling Code".ROB3_Unloading_Robot.Gripper."SHAFT CLAMPING RIGHT" := 'SZ23055-OP010-E-Compressor-robot3 shaft Right clamping jaw tooling-2';
   PRODUCT_TYPE[10]."Tooling Code".A1_Fixtures.A1RingUnloadingFixtureCode := 'SZ23055-OP010-E-Compresspr-ring1 cutting tool';
   PRODUCT_TYPE[10]."Tooling Code".A1_Fixtures.E1LoadingNGFixtureCode := 'SZ23055-OP010-E-Compressor-Left NG tooling-1';
   PRODUCT_TYPE[10]."Tooling Code".A1_Fixtures.ShaftScanFixtureCode := 'SZ23055-OP010-E-Compressor-shaft Rotating scanning tooling-1';
   PRODUCT_TYPE[10]."Tooling Code".A1_Fixtures.B1PressFixtureCode := 'SZ23055-OP010-E-Compressor-ring1 Below Positioning fixture -1';
   PRODUCT_TYPE[10]."Tooling Code".A1_Fixtures.CGlueFixtureCode := 'SZ23055-OP010-E-Compressor-Point adhesive tooling-1';
   PRODUCT_TYPE[10]."Tooling Code".A1_Fixtures.B1PressCylFixtureCode := 'SZ23055-OP010-E-Compressor-ring1 Upper pressing fixture-1';
   PRODUCT_TYPE[10]."Tooling Code".A2_Fixtures.A2RingUnloadingFixtureCode := 'SZ23055-OP010-E-Compresspr-ring2 cutting tool';
   PRODUCT_TYPE[10]."Tooling Code".A2_Fixtures.E2UnloadingNGFixtureCode := 'SZ23055-OP010-E-Compressor-Right NG tooling-1';
   PRODUCT_TYPE[10]."Tooling Code".A2_Fixtures.B2PressFixtureCode := 'SZ23055-OP010-E-Compressor-ring2 Below Positioning fixture -1';
   PRODUCT_TYPE[10]."Tooling Code".A2_Fixtures.CGlueNGFixtureCode := 'SZ23055-OP010-E-Compressor-NG middle shift tooling-1';
   PRODUCT_TYPE[10]."Tooling Code".A2_Fixtures.B2PressCylFixtureCode := 'SZ23055-OP010-E-Compressor-ring2 Upper pressing fixture-1';

